(* PLC project CoDeSys External Library Template, WAGO e!COCKPIT e!COCKPIT, author 3S - Smart Software Solutions GmbH *)
(* stored: creationDateTime 2019-10-29T12:22:40.7336323, version 3.5.5.30, modificationDateTime 2019-10-24T14:40:07.960949, organization 3S - Smart Software Solutions GmbH *)
(* Library project template with all possible element types, docu and a sample project structure *)

FUNCTION_BLOCK fbPPPSWezelClimatixPOL63x
  VAR_INPUT
    sKomunikat : alSTRINGKomunikat;  (* komunikat z systemu zewnętrznego *)
    intTablicaKomunikatowRozmiar : INT;  (* rozmiar tablicy danych wysyłkowych *)
    intModbusOdczytZapisZadanieRozmiar : INT;  (* rozmiar tablicy danych modbusa *)
    xTablicaKomunikatowHold : BOOL;  (* wstrzymanie komunikacji mniej ważnych komunikatów *)
    sIdInstancji : STRING;  (* parametr ID rolety np NS02L*202IBM**** *)
    sIdAplikacji : STRING;  (* parametr ID aplikacji np SO*******ECL*000 *)
    sMnemonik : STRING;  (* mnemonik właściciela - BCB* *)
    sMACAdres : STRING;  (* MAC adres sterownika *)
    sDaneZapasowe : STRING;  (* 6 znaków zapasu *)
    tCzasOpoznieniaRestartu : TIME;  (* czas opóźnienia po którym zaczynają być raportowane wartości *)
    tCzasOpoznieniaAlarmu : TIME := TIME#1m0s0ms;  (* czas opóźnienia po którym zaczynają być raportowane wartości *)
    bAdres : BYTE;
    tMinimalnyCzasRaportowania : TIME;
    tMaksymalnyCzasRaportowania : TIME;
    xAutonomizacja : BOOL;
    xAutonomizacjaSztuczna : BOOL;
    xSezonGrzewczyCalyRok : BOOL;
    tCzestotliwoscWysylaniaAlternatywnyAlgorytm : TIME;
    wZaprogramowanyTypInstalacji : WORD;
    rKrzywaGrzewczaTemperaturyZewnetrznejX2HC1Autonomizacja : REAL;  (* Sterowanie w trybie autonomizacji *)
    rKrzywaGrzewczaTemperaturyZasilaniaY2HC1Autonomizacja : REAL;
    rKrzywaGrzewczaTemperaturyZewnetrznejX3HC1Autonomizacja : REAL;
    rKrzywaGrzewczaTemperaturyZasilaniaY3HC1Autonomizacja : REAL;
    rKrzywaGrzewczaTemperaturyZewnetrznejX4HC1Autonomizacja : REAL;
    rKrzywaGrzewczaTemperaturyZasilaniaY4HC1Autonomizacja : REAL;
    rKrzywaGrzewczaTemperaturyZewnetrznejX5HC1Autonomizacja : REAL;
    rKrzywaGrzewczaTemperaturyZasilaniaY5HC1Autonomizacja : REAL;
    rKrzywaGrzewczaTemperaturyZewnetrznejX6HC1Autonomizacja : REAL;
    rKrzywaGrzewczaTemperaturyZasilaniaY6HC1Autonomizacja : REAL;
    intTrybPracyDHWAutonomizacja : INT;
  END_VAR
  VAR_IN_OUT
    arModbusOdczytCykliczny : ARRAY[1..5000] OF typModbusOdczytCykliczny;
    arModbusStatusKomunikacji : ARRAY[1..256] OF INT;
    arModbusOdczytZapisZadanie : ARRAY[1..1000] OF typModbusOdczytZapisZadanie;
    intModbusOdczytZapisZadanieZnacznikZapisu : INT;
    arTablicaKomunikatow : alARRAYTablicaKomunikatow;
    intTablicaKomunikatowZnacznikZapisu : INT;
    aTemperatury : ARRAY[0..96] OF REAL;  (* Tablica pomiarów temperatur bieżącego dnia *)
    rTemperaturaSrednia1Dzien : REAL;  (* Średnia dzienna temperatura *)
    iTemperaturyIndex : INT;  (* Index tablicy *)
    aTemperaturySrednie : ARRAY[0..2] OF REAL;  (* Tablica zawierająca średnie temperatury z trzech ostatnich dni *)
    iTemperaturySrednieIndex : INT;  (* Index tablicy śrenich temperatur *)
    rTemperaturaSrednia3Dni : REAL;  (* Średnia temperatura z trzech dni *)
    xTemperaturaSrednia3DniObliczona : BOOL;  (* Prawda, jeśli obliczona została średnia temperatura z trzech dni *)
  END_VAR
  VAR CONSTANT
    uintTrybPracyHC1AdresModbus : UINT := 400;  (* 1 *)
    uintKrzywaGrzewczaTemperaturyZewnetrznejX2HC1AdresModbus : UINT := 424;  (* 2 *)
    uintKrzywaGrzewczaTemperaturyZewnetrznejX3HC1AdresModbus : UINT := 449;  (* 9 *)
    uintKrzywaGrzewczaTemperaturyZewnetrznejX4HC1AdresModbus : UINT := 450;  (* 10 *)
    uintKrzywaGrzewczaTemperaturyZewnetrznejX5HC1AdresModbus : UINT := 451;  (* 11 *)
    uintKrzywaGrzewczaTemperaturyZewnetrznejX6HC1AdresModbus : UINT := 425;  (* 3 *)
    uintKrzywaGrzewczaTemperaturyZasilaniaY2HC1AdresModbus : UINT := 426;  (* 4 *)
    uintKrzywaGrzewczaTemperaturyZasilaniaY3HC1AdresModbus : UINT := 435;  (* 6 *)
    uintKrzywaGrzewczaTemperaturyZasilaniaY4HC1AdresModbus : UINT := 436;  (* 7 *)
    uintKrzywaGrzewczaTemperaturyZasilaniaY5HC1AdresModbus : UINT := 437;  (* 8 *)
    uintKrzywaGrzewczaTemperaturyZasilaniaY6HC1AdresModbus : UINT := 427;  (* 5 *)
    uintTrybPracyZadanieDHWAdresModbus : UINT := 800;  (* 12 *)
  END_VAR
  VAR
    xPierwszySkan : BOOL := TRUE;
    intPetlaPierwszySkan : INT := 1;
    xInstalacjaHC1 : BOOL;  (* Heat circuit 1 - 1-szy obwód grzewczy *)
    xInstalacjaDHW : BOOL;  (* Domestic hot water - ciepła woda użytkowa *)
    xInstalacjaHP : BOOL;  (* ??? - BRAK ZAPROGRAMOWANIA *)
    xInstalacjaHC2 : BOOL;  (* Heat circuit 2 - 2-gi obwód grzewczy - BRAK ZAPROGRAMOWANIA *)
    fbAutonomizacja : R_TRIG;  (* Wykrywanie przejścia w stan autonomizacji *)
    xPrzywrocDomyslne : BOOL;  (* Przywrócenie nastaw krzywej grzewczej i trybów pracy (przepisanie rAutonomizacjaKrzywaGrzewcza[...] etc. do Climatixa) *)
    intBlokadaWykonywaniaRozkazow : INT;
    intBlokadaWykonywaniaRozkazowZaraportowana : INT;
    xOdczytanaKlasaAlarmuBezpieczenstwa : BOOL := FALSE;  (* definicja zmiennych do odczytu wartości z modbusa klasy alarmów *)
    xOdczytanaKlasaAlarmuKrytyczny : BOOL := FALSE;
    xOdczytanaKlasaAlarmuOstrzezenie : BOOL := FALSE;
    xOdczytanaKlasaAlarmuInformacyjny : BOOL := FALSE;
    wAlarmsWord1 : WORD;  (* alarmy *)
    wAlarmsWord1Zaraportowana : WORD;
    wAlarmsWord2 : WORD;
    wAlarmsWord2Zaraportowana : WORD;
    wAlarmsWord3 : WORD;
    wAlarmsWord3Zaraportowana : WORD;
    wAlarmsWord4 : WORD;
    wAlarmsWord4Zaraportowana : WORD;
    wActiveAlarmsClass0 : WORD;
    wActiveAlarmsClass1 : WORD;
    wActiveAlarmsClass2 : WORD;
    wActiveAlarmsClass3 : WORD;
    wReczneWylaczenieInstalacji : WORD;  (* odczyt *)
    xReczneWylaczenieInstalacji : BOOL;
    wTypInstalacji : WORD;  (* 0=Other,1=1 HC,2=1 HC + DHW,3=1 HC + DHW + HP,4=2 HC,5=2 HC + DHW,6=2 HC + DHW + HP,7=Free (other combination) *)
    wTemperaturaZewnetrzna : WORD;  (* HC1 Temperatura zewnętrzna *)
    rTemperaturaZewnetrzna : REAL;
    fbTemperaturaZewnetrzna : fbFiltrWartoscAnalogowa;
    rTemperaturaZewnetrznaZaraportowana : REAL;
    wTemperaturaGrzaniaNastawionaHC1 : WORD;  (* Temperatura nastawiona zasilania *)
    rTemperaturaGrzaniaNastawionaHC1 : REAL;
    fbTemperaturaGrzaniaNastawionaHC1 : fbFiltrWartoscAnalogowa;
    rTemperaturaGrzaniaNastawionaHC1Zaraportowana : REAL;
    wTemperaturaGrzaniaNastawionaKrzywaGrzewczaHC1 : WORD;  (* Temperatura nastawiona zasilania z krzywej grzewczej *)
    rTemperaturaGrzaniaNastawionaKrzywaGrzewczaHC1 : REAL;
    fbTemperaturaGrzaniaNastawionaKrzywaGrzewczaHC1 : fbFiltrWartoscAnalogowa;
    rTemperaturaGrzaniaNastawionaKrzywaGrzewczaHC1Zaraportowana : REAL;
    wTrybPracyHC1 : WORD;  (* Tryb Pracy *)
    intTrybPracyHC1 : INT;
    intTrybPracyHC1Zaraportowana : INT;
    intTrybPracyHC1Autonomizacja : INT;
    wTrybPracyHC1Ramka : WORD;
    xTrybPracyHC1Zapisz : BOOL;  (* Trigger zapisu wartości w pamięci urządzenia *)
    rTrybPracyHC1Zapis : REAL;  (* Wartość do zapisania w pamięci urządzenia *)
    wTrybOperacjiHC1 : WORD;  (* Tryb operacji *)
    intTrybOperacjiHC1 : INT;
    intTrybOperacjiHC1Zaraportowana : INT;
    wTemperaturaZasilaniaObwoduHC1 : WORD;  (* Obwód na instalację *)
    rTemperaturaZasilaniaObwoduHC1 : REAL;
    fbTemperaturaZasilaniaObwoduHC1 : fbFiltrWartoscAnalogowa;
    rTemperaturaZasilaniaObwoduHC1Zaraportowana : REAL;
    wTemperaturaPowrotuObwoduHC1 : WORD;  (* Obwód na instalację *)
    rTemperaturaPowrotuObwoduHC1 : REAL;
    fbTemperaturaPowrotuObwoduHC1 : fbFiltrWartoscAnalogowa;
    rTemperaturaPowrotuObwoduHC1Zaraportowana : REAL;
    wTemperaturaPowrotuMiastoHC1 : WORD;  (* Powrót przy wymienniku ciepła po stronie wyskoiego parametru (miejskiej sieci ciepłowniczej) *)
    rTemperaturaPowrotuMiastoHC1 : REAL;
    fbTemperaturaPowrotuMiastoHC1 : fbFiltrWartoscAnalogowa;
    rTemperaturaPowrotuMiastoHC1Zaraportowana : REAL;
    wTemperaturaZasilaniaBudynku : WORD;  (* Zasilanie przy wymienniku ciepła po stronie budynku *)
    rTemperaturaZasilaniaBudynku : REAL;
    fbTemperaturaZasilaniaBudynku : fbFiltrWartoscAnalogowa;
    rTemperaturaZasilaniaBudynkuZaraportowana : REAL;
    wTemperaturaPowrotuBudynku : WORD;  (* Powrót przy wymienniku ciepła po stronie budynku *)
    rTemperaturaPowrotuBudynku : REAL;
    fbTemperaturaPowrotuBudynku : fbFiltrWartoscAnalogowa;
    rTemperaturaPowrotuBudynkuZaraportowana : REAL;
    wSygnalZadaniaGrzaniaHC1 : WORD;  (* Sygnał żądanego grzania, w procentach *)
    rSygnalZadaniaGrzaniaHC1 : REAL;
    fbSygnalZadaniaGrzaniaHC1 : fbFiltrWartoscAnalogowa;
    rSygnalZadaniaGrzaniaHC1Zaraportowana : REAL;
    wStopienOtwarciaZaworuMiastoHC1 : WORD;  (* Stopień otwarcia zaworu na powrocie wymiennika po stronie miejskiej sieci ciepłowniczej *)
    rStopienOtwarciaZaworuMiastoHC1 : REAL;
    fbStopienOtwarciaZaworuMiastoHC1 : fbFiltrWartoscAnalogowa;
    rStopienOtwarciaZaworuMiastoHC1Zaraportowana : REAL;
    wKrzywaGrzewczaTemperaturyZewnetrznejX2OdczytHC1 : WORD;  (* Krzywa grzewcza X2 *)
    rKrzywaGrzewczaTemperaturyZewnetrznejX2HC1 : REAL;
    fbKrzywaGrzewczaTemperaturyZewnetrznejX2HC1 : fbFiltrWartoscAnalogowa;
    rKrzywaGrzewczaTemperaturyZewnetrznejX2HC1Zaraportowana : REAL;
    xKrzywaGrzewczaTemperaturyZewnetrznejX2HC1Zapisz : BOOL;  (* Trigger zapisu wartości w pamięci urządzenia *)
    rKrzywaGrzewczaTemperaturyZewnetrznejX2HC1Zapis : REAL;  (* Wartość do zapisania w pamięci urządzenia *)
    wKrzywaGrzewczaTemperaturyZewnetrznejX2HC1Zapis : WORD;  (* Wartość do zapisania w pamięci urządzenia (po konwersji na WORDa) *)
    rKrzywaGrzewczaTemperaturyZewnetrznejX2HC1Raport : REAL;  (* Wartość do zaraportowania *)
    wKrzywaGrzewczaTemperaturyZasilaniaY2OdczytHC1 : WORD;  (* Krzywa grzewcza Y2 *)
    rKrzywaGrzewczaTemperaturyZasilaniaY2HC1 : REAL;
    fbKrzywaGrzewczaTemperaturyZasilaniaY2HC1 : fbFiltrWartoscAnalogowa;
    rKrzywaGrzewczaTemperaturyZasilaniaY2HC1Zaraportowana : REAL;
    xKrzywaGrzewczaTemperaturyZasilaniaY2HC1Zapisz : BOOL;  (* Trigger zapisu wartości w pamięci urządzenia *)
    rKrzywaGrzewczaTemperaturyZasilaniaY2HC1Zapis : REAL;  (* Wartość do zapisania w pamięci urządzenia *)
    wKrzywaGrzewczaTemperaturyZewnetrznejX3OdczytHC1 : WORD;  (* Krzywa grzewcza X3 *)
    rKrzywaGrzewczaTemperaturyZewnetrznejX3HC1 : REAL;
    fbKrzywaGrzewczaTemperaturyZewnetrznejX3HC1 : fbFiltrWartoscAnalogowa;
    rKrzywaGrzewczaTemperaturyZewnetrznejX3HC1Zaraportowana : REAL;
    xKrzywaGrzewczaTemperaturyZewnetrznejX3HC1Zapisz : BOOL;  (* Trigger zapisu wartości w pamięci urządzenia *)
    rKrzywaGrzewczaTemperaturyZewnetrznejX3HC1Zapis : REAL;  (* Wartość do zapisania w pamięci urządzenia *)
    wKrzywaGrzewczaTemperaturyZewnetrznejX3HC1Zapis : WORD;  (* Wartość do zapisania w pamięci urządzenia (po konwersji na WORDa) *)
    rKrzywaGrzewczaTemperaturyZewnetrznejX3HC1Raport : REAL;  (* Wartość do zaraportowania *)
    wKrzywaGrzewczaTemperaturyZasilaniaY3OdczytHC1 : WORD;  (* Krzywa grzewcza Y3 *)
    rKrzywaGrzewczaTemperaturyZasilaniaY3HC1 : REAL;
    fbKrzywaGrzewczaTemperaturyZasilaniaY3HC1 : fbFiltrWartoscAnalogowa;
    rKrzywaGrzewczaTemperaturyZasilaniaY3HC1Zaraportowana : REAL;
    xKrzywaGrzewczaTemperaturyZasilaniaY3HC1Zapisz : BOOL;  (* Trigger zapisu wartości w pamięci urządzenia *)
    rKrzywaGrzewczaTemperaturyZasilaniaY3HC1Zapis : REAL;  (* Wartość do zapisania w pamięci urządzenia *)
    wKrzywaGrzewczaTemperaturyZewnetrznejX4OdczytHC1 : WORD;  (* Krzywa grzewcza X4 *)
    rKrzywaGrzewczaTemperaturyZewnetrznejX4HC1 : REAL;
    fbKrzywaGrzewczaTemperaturyZewnetrznejX4HC1 : fbFiltrWartoscAnalogowa;
    rKrzywaGrzewczaTemperaturyZewnetrznejX4HC1Zaraportowana : REAL;
    xKrzywaGrzewczaTemperaturyZewnetrznejX4HC1Zapisz : BOOL;  (* Trigger zapisu wartości w pamięci urządzenia *)
    rKrzywaGrzewczaTemperaturyZewnetrznejX4HC1Zapis : REAL;  (* Wartość do zapisania w pamięci urządzenia *)
    wKrzywaGrzewczaTemperaturyZewnetrznejX4HC1Zapis : WORD;  (* Wartość do zapisania w pamięci urządzenia (po konwersji na WORDa) *)
    rKrzywaGrzewczaTemperaturyZewnetrznejX4HC1Raport : REAL;  (* Wartość do zaraportowania *)
    wKrzywaGrzewczaTemperaturyZasilaniaY4OdczytHC1 : WORD;  (* Krzywa grzewcza Y4 *)
    rKrzywaGrzewczaTemperaturyZasilaniaY4HC1 : REAL;
    fbKrzywaGrzewczaTemperaturyZasilaniaY4HC1 : fbFiltrWartoscAnalogowa;
    rKrzywaGrzewczaTemperaturyZasilaniaY4HC1Zaraportowana : REAL;
    xKrzywaGrzewczaTemperaturyZasilaniaY4HC1Zapisz : BOOL;  (* Trigger zapisu wartości w pamięci urządzenia *)
    rKrzywaGrzewczaTemperaturyZasilaniaY4HC1Zapis : REAL;  (* Wartość do zapisania w pamięci urządzenia *)
    wKrzywaGrzewczaTemperaturyZewnetrznejX5OdczytHC1 : WORD;  (* Krzywa grzewcza X5 *)
    rKrzywaGrzewczaTemperaturyZewnetrznejX5HC1 : REAL;
    fbKrzywaGrzewczaTemperaturyZewnetrznejX5HC1 : fbFiltrWartoscAnalogowa;
    rKrzywaGrzewczaTemperaturyZewnetrznejX5HC1Zaraportowana : REAL;
    xKrzywaGrzewczaTemperaturyZewnetrznejX5HC1Zapisz : BOOL;  (* Trigger zapisu wartości w pamięci urządzenia *)
    rKrzywaGrzewczaTemperaturyZewnetrznejX5HC1Zapis : REAL;  (* Wartość do zapisania w pamięci urządzenia *)
    wKrzywaGrzewczaTemperaturyZewnetrznejX5HC1Zapis : WORD;  (* Wartość do zapisania w pamięci urządzenia (po konwersji na WORDa) *)
    rKrzywaGrzewczaTemperaturyZewnetrznejX5HC1Raport : REAL;  (* Wartość do zaraportowania *)
    wKrzywaGrzewczaTemperaturyZasilaniaY5OdczytHC1 : WORD;  (* Krzywa grzewcza Y5 *)
    rKrzywaGrzewczaTemperaturyZasilaniaY5HC1 : REAL;
    fbKrzywaGrzewczaTemperaturyZasilaniaY5HC1 : fbFiltrWartoscAnalogowa;
    rKrzywaGrzewczaTemperaturyZasilaniaY5HC1Zaraportowana : REAL;
    xKrzywaGrzewczaTemperaturyZasilaniaY5HC1Zapisz : BOOL;  (* Trigger zapisu wartości w pamięci urządzenia *)
    rKrzywaGrzewczaTemperaturyZasilaniaY5HC1Zapis : REAL;  (* Wartość do zapisania w pamięci urządzenia *)
    wKrzywaGrzewczaTemperaturyZewnetrznejX6OdczytHC1 : WORD;  (* Krzywa grzewcza X6 *)
    rKrzywaGrzewczaTemperaturyZewnetrznejX6HC1 : REAL;
    fbKrzywaGrzewczaTemperaturyZewnetrznejX6HC1 : fbFiltrWartoscAnalogowa;
    rKrzywaGrzewczaTemperaturyZewnetrznejX6HC1Zaraportowana : REAL;
    xKrzywaGrzewczaTemperaturyZewnetrznejX6HC1Zapisz : BOOL;  (* Trigger zapisu wartości w pamięci urządzenia *)
    rKrzywaGrzewczaTemperaturyZewnetrznejX6HC1Zapis : REAL;  (* Wartość do zapisania w pamięci urządzenia *)
    wKrzywaGrzewczaTemperaturyZewnetrznejX6HC1Zapis : WORD;  (* Wartość do zapisania w pamięci urządzenia (po konwersji na WORDa) *)
    rKrzywaGrzewczaTemperaturyZewnetrznejX6HC1Raport : REAL;  (* Wartość do zaraportowania *)
    wKrzywaGrzewczaTemperaturyZasilaniaY6OdczytHC1 : WORD;  (* Krzywa grzewcza Y6 *)
    rKrzywaGrzewczaTemperaturyZasilaniaY6HC1 : REAL;
    fbKrzywaGrzewczaTemperaturyZasilaniaY6HC1 : fbFiltrWartoscAnalogowa;
    rKrzywaGrzewczaTemperaturyZasilaniaY6HC1Zaraportowana : REAL;
    xKrzywaGrzewczaTemperaturyZasilaniaY6HC1Zapisz : BOOL;  (* Trigger zapisu wartości w pamięci urządzenia *)
    rKrzywaGrzewczaTemperaturyZasilaniaY6HC1Zapis : REAL;  (* Wartość do zapisania w pamięci urządzenia *)
    wTemperaturaGrzaniaNastawionaDHW : WORD;  (* DHW Temperatura nastawiona zasilania *)
    rTemperaturaGrzaniaNastawionaDHW : REAL;
    fbTemperaturaGrzaniaNastawionaDHW : fbFiltrWartoscAnalogowa;
    rTemperaturaGrzaniaNastawionaDHWZaraportowana : REAL;
    wTrybPracyDHW : WORD;  (* Tryb Pracy *)
    intTrybPracyDHW : INT;
    intTrybPracyDHWZaraportowana : INT;
    wTrybPracyDHWRamka : WORD;
    xTrybPracyDHWZapisz : BOOL;  (* Trigger zapisu wartości w pamięci urządzenia *)
    rTrybPracyDHWZapis : REAL;  (* Wartość do zapisania w pamięci urządzenia *)
    wTrybOperacjiDHW : WORD;  (* Tryb operacji *)
    intTrybOperacjiDHW : INT;
    intTrybOperacjiDHWZaraportowana : INT;
    wTemperaturaPowrotuMiastoDHW : WORD;  (* Powrót przy wymienniku ciepła po stronie wyskoiego parametru (miejskiej sieci ciepłowniczej) *)
    rTemperaturaPowrotuMiastoDHW : REAL;
    fbTemperaturaPowrotuMiastoDHW : fbFiltrWartoscAnalogowa;
    rTemperaturaPowrotuMiastoDHWZaraportowana : REAL;
    wTemperaturaZasilaniaBudynekDHW : WORD;  (* Zasilanie przy wymienniku ciepła po stronie budynku *)
    rTemperaturaZasilaniaBudynekDHW : REAL;
    fbTemperaturaZasilaniaBudynekDHW : fbFiltrWartoscAnalogowa;
    rTemperaturaZasilaniaBudynekDHWZaraportowana : REAL;
    wTemperaturaPowrotuBudynekDHW : WORD;  (* Powrót przy wymienniku ciepła po stronie budynku *)
    rTemperaturaPowrotuBudynekDHW : REAL;
    fbTemperaturaPowrotuBudynekDHW : fbFiltrWartoscAnalogowa;
    rTemperaturaPowrotuBudynekDHWZaraportowana : REAL;
    wStopienOtwarciaZaworuMiastoDHW : WORD;  (* Stopień otwarcia zaworu na powrocie wymiennika po stronie miejskiej sieci ciepłowniczej *)
    rStopienOtwarciaZaworuMiastoDHW : REAL;
    fbStopienOtwarciaZaworuMiastoDHW : fbFiltrWartoscAnalogowa;
    rStopienOtwarciaZaworuMiastoDHWZaraportowana : REAL;
    xPoInicjalizacji : BOOL := FALSE;  (* inicjalizacja *)
    fbInicjalizacyjnyTimer : TON;
    tCzasInicjalizacji : TIME := TIME#30s0ms;
    sDane : alSTRINGKomunikat;  (* pozostale definicje *)
    sWyslanyKomunikatDummy : alSTRINGKomunikat;
    xZadanieRaportu : BOOL;
    sKomunikatPamiec : alSTRINGKomunikat;
    intPetla : INT;
    arErrorStan : ARRAY[0..11] OF INT;  (* tablica przechowująca statusy alarmowe *)
    arErrorKlasa : ARRAY[0..11] OF INT;  (* tablica przechowująca klasy danych alarmów *)
    xRaport : BOOL := FALSE;
    sTempWartoscAtrybutu : STRING;
    xOverFlow : BOOL;
    rtrigPrzywrocDomyslne : R_TRIG;  (* Przywracanie domyślnych wartości nastaw *)
    rtrigZapisModbus : R_TRIG;  (* Triger zapisu danych po Modbusie *)
    fbTaktowanieZapisywaniaModbus : TON;  (* Cykliczne żądanie zapisu danych do urządzenia *)
    fbTimerBrakuKomunikacji : TON;  (* Kontrola komunikacji urządzenia *)
    xBrakKomunikacjiPLC : BOOL;
    xBrakKomunikacjiIZE : BOOL;
    wTrybPracyZadanie : INT;
    rAutonomizacjaKorektaTemperaturyGrzaniaZadanie : INT;
    xBrakKomunikacji : BOOL;
    rTemperaturaZewnetrznaPamiec : REAL;  (* Sprawdzanie sprawności czujnika temperatury zewnętrznej *)
    xBrakZmianyTemperaturyZewnetrznej : BOOL;
    fbBrakZmianyTemperaturyZewnetrznejTimer : TON;
    xBladBrakZmianyTemperaturyZewnetrznej : BOOL;
    rTemperaturaZasilaniaObwoduHC1Pamiec : REAL;  (* Sprawdzanie sprawności czujnika temperatury zasilania obwodu HC1 *)
    xBrakZmianyTemperaturyZasilaniaObwoduHC1 : BOOL;
    fbBrakZmianyTemperaturyZasilaniaObwoduHC1Timer : TON;
    xBladBrakZmianyTemperaturyZasilaniaObwoduHC1 : BOOL;
    rTemperaturaZasilaniaObwoduDHWPamiec : REAL;  (* Sprawdzanie sprawności czujnika temperatury zasilania obwodu DHW *)
    xBrakZmianyTemperaturyZasilaniaObwoduDHW : BOOL;
    fbBrakZmianyTemperaturyZasilaniaObwoduDHWTimer : TON;
    xBladBrakZmianyTemperaturyZasilaniaObwoduDHW : BOOL;
    xBrakOsiagnieciaTemperauryZadanejHC1 : BOOL;  (* Sprawdzanie czy została osiągnęta zadana temperatura zasilania obwodu HC1 *)
    fbBrakOsiagnieciaTemperauryZadanejHC1Timer : TON;
    xBladBrakOsiagnieciaTemperauryZadanejHC1 : BOOL;
    xBrakOsiagnieciaTemperauryZadanejDHW : BOOL;  (* Sprawdzanie czy została osiągnęta zadana temperatura zasilania obwodu DHW *)
    fbBrakOsiagnieciaTemperauryZadanejDHWTimer : TON;
    xBladBrakOsiagnieciaTemperauryZadanejDHW : BOOL;
    fbWschodZachod : FbCalculateSunriseSunset;  (* Obliczanie wschodu i zachodu słońca *)
    fbZegar15M : TON;  (* Timer taktujący zapisywanie temperatury *)
    xObliczSrednia3Dni : BOOL;  (* Triger obliczania średniej dziennej temperatury z 3 ostatnich dni *)
    iIloscPomiarow : INT;  (* Ilość pomiarów dokonanych w ciągu dnia *)
    rTemperaturaSrednia1DzienZaraportowana : REAL;  (* Średnia dzienna temperatura zaraporotawana *)
    xSezonGrzewczy : BOOL;  (* Włączenie ogrzewania *)
    xSezonGrzewczyZaraportowana : BOOL;  (* Włączenie ogrzewania zaraportowane *)
    xBladIloscPomiarowTemperatury : BOOL;  (* Zbyt mała ilość pomiarów dokonanych w ciągu dnia do obliczenia średniej *)
  END_VAR

            (*			
Autor:					Paweł Kąkol, 2018-09-03 
Prawa majątkowe: 		Solwena Sp. z o.o., 
Aktualizacje:			2018-09-06-PK: zmiana adresów rejestrów o -1
						2018-09-07-PK: przerobienie całego fb tak aby realizował układ HC1 (1-szego obiegu grzewczego) oraz/lub DHW (ciepłej wody użytkowej), wykonanie reakcji na autonomizację
						2019-01-04-AW: zmiana odczytu klasy alarmów (zmiana funkcji i adresów); odczyt rejestrów zawierających info o rodzaju alarmu
						2019-02-08-AWy: OverFlow
						2019-02-10-AWy: odczyt trybu operacji HC1 i wysyłanie do IZE, poprawa odczytywania i wysyłania temperatury zasilania, powrotu obwodu i miasta, krzywej grzewczej etc.
						2019-02-18-AWy: odczyt trybu operacji DHW i wysyłanie do IZE
						2019-05-15-AWy: - modyfikacja warunku obsługi ramki C. Było: IF sTempWartoscAtrybutu <> '' AND intBlokadaWykonywaniaRozkazow = 0 THEN. Jest: IF intBlokadaWykonywaniaRozkazow = 0 THEN
						2019-05-16-AWy: - modyfikacja warunku ręcznej inizjalizacji trybów pracy i krzywej grzewczej. Było: IF xAutonomizacja THEN. Jest: IF xPrzywrocDomyslne THEN.
									    - modyfikacja warunku na raportowanie. Dopisane: AND xPoInicjalizacji
									    - modyfikacja warunków na zapis po otrzymaniu ramki C. Nowy warunek: IF fnKomunikatDaneSzukajWartosci(sKomunikat,'TEMPKGHC1X5=') <> '' THEN etc.
						2019-05-23-AWy: dodanie przesyłania wewnętrznych numerów błędów z Climatixa (wAlarmsWord1 etc.)
						2019-06-03-AWy: załadowanie domyślnych trybów pracy i nastaw po przejściu w tryb autonomizacji
						2019-06-04-AWy: usunięcie błędów generowanych przy odczycie liczb ujemnych
						2019-07-16-AWy: zmiana typu zmiennej intTrybPracyDHWAutonomizacja z WORD na INT
						2019-08-05-AWy: wyznaczanie okresu grzewczego. Wysyłanie xSezonGrzewczy i rTemperaturaSrednia1Dzien do IZE. Przeniesie xTrybPracyAutonomizacja z VAR_INPUT do VAR
						2019-10-22-AWy: - wydłużenie czasu fbTaktowanieZapisywaniaModbus oraz wprowadzenie trigera zapisu po Modbusie
										- zmiana trigera fbTimerBrakuKomunikacji
						
Opis:					fb służy do komunikacji po Modbus RTU z węzłem ciepła na budynkach ENGIE, gdzie zainstalowano Siemens Climatix POL638.70
						Zawiera kod wykonywany w razie autonomizacji - wysyłanie zmiennych wprowadzonych poprzez EIG,
						po ustaniu Autonomizacji zostaje utrzymany stan z Autonomizacji, a układ reaguje dopiero na nowe ramki

UWAGA:					Zaprogramowano HC1 oraz DHN, nie zaprogramowane HP i HC2 
*)


//inicjalizacja sterownika
fbInicjalizacyjnyTimer(IN := (NOT xPoInicjalizacji AND arModbusStatusKomunikacji[bAdres] = enumModbusStatus.KomunikacjaPrawidlowa) , PT := tCzasOpoznieniaRestartu);
IF fbInicjalizacyjnyTimer.Q THEN
	IF xInstalacjaHC1 OR xInstalacjaHC2 THEN
		rTemperaturaZewnetrznaZaraportowana := rTemperaturaZewnetrzna;
	END_IF
	IF xInstalacjaHC1 THEN
		rTemperaturaGrzaniaNastawionaHC1Zaraportowana := rTemperaturaGrzaniaNastawionaHC1;
		rTemperaturaGrzaniaNastawionaKrzywaGrzewczaHC1Zaraportowana := rTemperaturaGrzaniaNastawionaKrzywaGrzewczaHC1;
		intTrybPracyHC1Zaraportowana := intTrybPracyHC1;
		intTrybOperacjiHC1 := intTrybOperacjiHC1Zaraportowana;
		rTemperaturaZasilaniaObwoduHC1Zaraportowana := rTemperaturaZasilaniaObwoduHC1;
		rTemperaturaPowrotuObwoduHC1Zaraportowana := rTemperaturaPowrotuObwoduHC1;
		rTemperaturaPowrotuMiastoHC1Zaraportowana := rTemperaturaPowrotuMiastoHC1;
		rTemperaturaZasilaniaBudynkuZaraportowana := rTemperaturaZasilaniaBudynku;
		rTemperaturaPowrotuBudynkuZaraportowana := rTemperaturaPowrotuBudynku;
		rSygnalZadaniaGrzaniaHC1Zaraportowana := rSygnalZadaniaGrzaniaHC1;
		rStopienOtwarciaZaworuMiastoHC1Zaraportowana := rStopienOtwarciaZaworuMiastoHC1;
		rKrzywaGrzewczaTemperaturyZewnetrznejX2HC1Zaraportowana := rKrzywaGrzewczaTemperaturyZewnetrznejX2HC1;
		rKrzywaGrzewczaTemperaturyZasilaniaY2HC1Zaraportowana := rKrzywaGrzewczaTemperaturyZasilaniaY2HC1;
		rKrzywaGrzewczaTemperaturyZewnetrznejX3HC1Zaraportowana := rKrzywaGrzewczaTemperaturyZewnetrznejX3HC1;
		rKrzywaGrzewczaTemperaturyZasilaniaY3HC1Zaraportowana := rKrzywaGrzewczaTemperaturyZasilaniaY3HC1;
		rKrzywaGrzewczaTemperaturyZewnetrznejX4HC1Zaraportowana := rKrzywaGrzewczaTemperaturyZewnetrznejX4HC1;
		rKrzywaGrzewczaTemperaturyZasilaniaY4HC1Zaraportowana := rKrzywaGrzewczaTemperaturyZasilaniaY4HC1;
		rKrzywaGrzewczaTemperaturyZewnetrznejX5HC1Zaraportowana := rKrzywaGrzewczaTemperaturyZewnetrznejX5HC1;
		rKrzywaGrzewczaTemperaturyZasilaniaY5HC1Zaraportowana := rKrzywaGrzewczaTemperaturyZasilaniaY5HC1;
		rKrzywaGrzewczaTemperaturyZewnetrznejX6HC1Zaraportowana := rKrzywaGrzewczaTemperaturyZewnetrznejX6HC1;
		rKrzywaGrzewczaTemperaturyZasilaniaY6HC1Zaraportowana := rKrzywaGrzewczaTemperaturyZasilaniaY6HC1;
		xSezonGrzewczyZaraportowana := xSezonGrzewczy;
		rTemperaturaSrednia1DzienZaraportowana := rTemperaturaSrednia1Dzien;
	END_IF
	IF xInstalacjaDHW THEN
		rTemperaturaGrzaniaNastawionaDHWZaraportowana := rTemperaturaGrzaniaNastawionaDHW;
		intTrybPracyDHWZaraportowana := intTrybPracyDHW;
		rTemperaturaPowrotuMiastoDHWZaraportowana := rTemperaturaPowrotuMiastoDHW;
		rTemperaturaZasilaniaBudynekDHWZaraportowana := rTemperaturaZasilaniaBudynekDHW;
		rTemperaturaPowrotuBudynekDHWZaraportowana := rTemperaturaPowrotuBudynekDHW;
		rStopienOtwarciaZaworuMiastoDHWZaraportowana := rStopienOtwarciaZaworuMiastoDHW;
		intTrybOperacjiDHWZaraportowana := intTrybOperacjiDHW;
	END_IF
	wAlarmsWord1Zaraportowana := wAlarmsWord1;
	wAlarmsWord2Zaraportowana := wAlarmsWord2;
	wAlarmsWord3Zaraportowana := wAlarmsWord3;
	wAlarmsWord4Zaraportowana := wAlarmsWord4;
	xPoInicjalizacji := TRUE;
END_IF

// Włącz autonomizację jeśli sterownik jest w stanie inicjalizacji lub nastąpiło wymuszenie autonomizacji
IF NOT xPoInicjalizacji OR xAutonomizacjaSztuczna = TRUE THEN
	xAutonomizacja := TRUE;
END_IF 

// Kontrola komunikacji
fbTimerBrakuKomunikacji(IN := arModbusStatusKomunikacji[bAdres] <> enumModbusStatus.KomunikacjaPrawidlowa, PT := T#60S);
IF fbTimerBrakuKomunikacji.Q THEN
	xBrakKomunikacjiPLC := TRUE;
ELSE
	xBrakKomunikacjiPLC := FALSE;
END_IF

IF xAutonomizacja THEN
	xBrakKomunikacjiIZE := TRUE;
ELSE
	xBrakKomunikacjiIZE := FALSE;
END_IF

// Deklaracja rejestrów Modbusa
IF xPierwszySkan THEN
	xPierwszySkan := FALSE;
	WHILE arModbusOdczytCykliczny[intPetlaPierwszySkan].bAdresUrzadzenia <> 0 DO
		intPetlaPierwszySkan := intPetlaPierwszySkan + 1;
	END_WHILE
	
	//wybrana instalacja na budynku
	CASE wZaprogramowanyTypInstalacji OF
		0:	xInstalacjaHC1 := FALSE;
			xInstalacjaDHW := FALSE;
			xInstalacjaHP := FALSE;
			xInstalacjaHC2 := FALSE;
		1:	xInstalacjaHC1 := TRUE;
			xInstalacjaDHW := FALSE;
			xInstalacjaHP := FALSE;
			xInstalacjaHC2 := FALSE;
		2:	xInstalacjaHC1 := TRUE;
			xInstalacjaDHW := TRUE;
			xInstalacjaHP := FALSE;
			xInstalacjaHC2 := FALSE;
		3:	xInstalacjaHC1 := TRUE;
			xInstalacjaDHW := TRUE;
			xInstalacjaHP := TRUE;
			xInstalacjaHC2 := FALSE;
		4:	xInstalacjaHC1 := TRUE;
			xInstalacjaDHW := FALSE;
			xInstalacjaHP := FALSE;
			xInstalacjaHC2 := TRUE;
		5:	xInstalacjaHC1 := TRUE;
			xInstalacjaDHW := TRUE;
			xInstalacjaHP := FALSE;
			xInstalacjaHC2 := TRUE;
		6:	xInstalacjaHC1 := TRUE;
			xInstalacjaDHW := TRUE;
			xInstalacjaHP := TRUE;
			xInstalacjaHC2 := TRUE;
	END_CASE
	
//deklaracja rejestrow do odczytu
	// Rejestry zawierające informację alarmach
	arModbusOdczytCykliczny[intPetlaPierwszySkan].bAdresUrzadzenia := bAdres;
	arModbusOdczytCykliczny[intPetlaPierwszySkan].bFunkcja := TO_BYTE(enumModbusKodyFunkcji.OdczytNRejestrowWejsciowych);
	arModbusOdczytCykliczny[intPetlaPierwszySkan].uiAdresRejestru := 18;
	arModbusOdczytCykliczny[intPetlaPierwszySkan].ltCzestotliwosc := LTIME#10S;
	arModbusOdczytCykliczny[intPetlaPierwszySkan].pZmiennaReferencyjna := ADR(wAlarmsWord1);
	intPetlaPierwszySkan := intPetlaPierwszySkan + 1;
	
	arModbusOdczytCykliczny[intPetlaPierwszySkan].bAdresUrzadzenia := bAdres;
	arModbusOdczytCykliczny[intPetlaPierwszySkan].bFunkcja := TO_BYTE(enumModbusKodyFunkcji.OdczytNRejestrowWejsciowych);
	arModbusOdczytCykliczny[intPetlaPierwszySkan].uiAdresRejestru := 19;
	arModbusOdczytCykliczny[intPetlaPierwszySkan].ltCzestotliwosc := LTIME#10S;
	arModbusOdczytCykliczny[intPetlaPierwszySkan].pZmiennaReferencyjna := ADR(wAlarmsWord2);
	intPetlaPierwszySkan := intPetlaPierwszySkan + 1;
	
	arModbusOdczytCykliczny[intPetlaPierwszySkan].bAdresUrzadzenia := bAdres;
	arModbusOdczytCykliczny[intPetlaPierwszySkan].bFunkcja := TO_BYTE(enumModbusKodyFunkcji.OdczytNRejestrowWejsciowych);
	arModbusOdczytCykliczny[intPetlaPierwszySkan].uiAdresRejestru := 20;
	arModbusOdczytCykliczny[intPetlaPierwszySkan].ltCzestotliwosc := LTIME#10S;
	arModbusOdczytCykliczny[intPetlaPierwszySkan].pZmiennaReferencyjna := ADR(wAlarmsWord3);
	intPetlaPierwszySkan := intPetlaPierwszySkan + 1;
	
	arModbusOdczytCykliczny[intPetlaPierwszySkan].bAdresUrzadzenia := bAdres;
	arModbusOdczytCykliczny[intPetlaPierwszySkan].bFunkcja := TO_BYTE(enumModbusKodyFunkcji.OdczytNRejestrowWejsciowych);
	arModbusOdczytCykliczny[intPetlaPierwszySkan].uiAdresRejestru := 21;
	arModbusOdczytCykliczny[intPetlaPierwszySkan].ltCzestotliwosc := LTIME#10S;
	arModbusOdczytCykliczny[intPetlaPierwszySkan].pZmiennaReferencyjna := ADR(wAlarmsWord4);
	intPetlaPierwszySkan := intPetlaPierwszySkan + 1;
	
	arModbusOdczytCykliczny[intPetlaPierwszySkan].bAdresUrzadzenia := bAdres;
	arModbusOdczytCykliczny[intPetlaPierwszySkan].bFunkcja := TO_BYTE(enumModbusKodyFunkcji.OdczytNRejestrowWejsciowych);
	arModbusOdczytCykliczny[intPetlaPierwszySkan].uiAdresRejestru := 22;
	arModbusOdczytCykliczny[intPetlaPierwszySkan].ltCzestotliwosc := LTIME#10S;
	arModbusOdczytCykliczny[intPetlaPierwszySkan].pZmiennaReferencyjna := ADR(wActiveAlarmsClass0);
	intPetlaPierwszySkan := intPetlaPierwszySkan + 1;
	
	arModbusOdczytCykliczny[intPetlaPierwszySkan].bAdresUrzadzenia := bAdres;
	arModbusOdczytCykliczny[intPetlaPierwszySkan].bFunkcja := TO_BYTE(enumModbusKodyFunkcji.OdczytNRejestrowWejsciowych);
	arModbusOdczytCykliczny[intPetlaPierwszySkan].uiAdresRejestru := 23;
	arModbusOdczytCykliczny[intPetlaPierwszySkan].ltCzestotliwosc := LTIME#10S;
	arModbusOdczytCykliczny[intPetlaPierwszySkan].pZmiennaReferencyjna := ADR(wActiveAlarmsClass1);
	intPetlaPierwszySkan := intPetlaPierwszySkan + 1;
	
	arModbusOdczytCykliczny[intPetlaPierwszySkan].bAdresUrzadzenia := bAdres;
	arModbusOdczytCykliczny[intPetlaPierwszySkan].bFunkcja := TO_BYTE(enumModbusKodyFunkcji.OdczytNRejestrowWejsciowych);
	arModbusOdczytCykliczny[intPetlaPierwszySkan].uiAdresRejestru := 24;
	arModbusOdczytCykliczny[intPetlaPierwszySkan].ltCzestotliwosc := LTIME#10S;
	arModbusOdczytCykliczny[intPetlaPierwszySkan].pZmiennaReferencyjna := ADR(wActiveAlarmsClass2);
	intPetlaPierwszySkan := intPetlaPierwszySkan + 1;
	
	arModbusOdczytCykliczny[intPetlaPierwszySkan].bAdresUrzadzenia := bAdres;
	arModbusOdczytCykliczny[intPetlaPierwszySkan].bFunkcja := TO_BYTE(enumModbusKodyFunkcji.OdczytNRejestrowWejsciowych);
	arModbusOdczytCykliczny[intPetlaPierwszySkan].uiAdresRejestru := 25;
	arModbusOdczytCykliczny[intPetlaPierwszySkan].ltCzestotliwosc := LTIME#10S;
	arModbusOdczytCykliczny[intPetlaPierwszySkan].pZmiennaReferencyjna := ADR(wActiveAlarmsClass3);
	intPetlaPierwszySkan := intPetlaPierwszySkan + 1;
	
	// Flagi typów alarmów (nie ma pewności, że działa - najprawdopodobniej w dokumentacji jest błąd i typy alarmów to nie inputy a coile - do zweryfikowania) - CAŁOŚĆ DO PRZETESTOWANIA
	arModbusOdczytCykliczny[intPetlaPierwszySkan].bAdresUrzadzenia := bAdres;
	arModbusOdczytCykliczny[intPetlaPierwszySkan].bFunkcja := TO_BYTE(enumModbusKodyFunkcji.OdczytWyjscBitowych);
	arModbusOdczytCykliczny[intPetlaPierwszySkan].uiAdresRejestru := 0;
	arModbusOdczytCykliczny[intPetlaPierwszySkan].ltCzestotliwosc := LTIME#10S;
	arModbusOdczytCykliczny[intPetlaPierwszySkan].pZmiennaReferencyjna := ADR(xOdczytanaKlasaAlarmuBezpieczenstwa);
	intPetlaPierwszySkan := intPetlaPierwszySkan + 1;		
	
	arModbusOdczytCykliczny[intPetlaPierwszySkan].bAdresUrzadzenia := bAdres;
	arModbusOdczytCykliczny[intPetlaPierwszySkan].bFunkcja := TO_BYTE(enumModbusKodyFunkcji.OdczytWyjscBitowych);
	arModbusOdczytCykliczny[intPetlaPierwszySkan].uiAdresRejestru := 1;
	arModbusOdczytCykliczny[intPetlaPierwszySkan].ltCzestotliwosc := LTIME#10S;
	arModbusOdczytCykliczny[intPetlaPierwszySkan].pZmiennaReferencyjna := ADR(xOdczytanaKlasaAlarmuKrytyczny);
	intPetlaPierwszySkan := intPetlaPierwszySkan + 1;	
	
	arModbusOdczytCykliczny[intPetlaPierwszySkan].bAdresUrzadzenia := bAdres;
	arModbusOdczytCykliczny[intPetlaPierwszySkan].bFunkcja := TO_BYTE(enumModbusKodyFunkcji.OdczytWyjscBitowych);
	arModbusOdczytCykliczny[intPetlaPierwszySkan].uiAdresRejestru := 2;
	arModbusOdczytCykliczny[intPetlaPierwszySkan].ltCzestotliwosc := LTIME#10S;
	arModbusOdczytCykliczny[intPetlaPierwszySkan].pZmiennaReferencyjna := ADR(xOdczytanaKlasaAlarmuOstrzezenie);
	intPetlaPierwszySkan := intPetlaPierwszySkan + 1;	
	
	arModbusOdczytCykliczny[intPetlaPierwszySkan].bAdresUrzadzenia := bAdres;
	arModbusOdczytCykliczny[intPetlaPierwszySkan].bFunkcja := TO_BYTE(enumModbusKodyFunkcji.OdczytWyjscBitowych);
	arModbusOdczytCykliczny[intPetlaPierwszySkan].uiAdresRejestru := 3;
	arModbusOdczytCykliczny[intPetlaPierwszySkan].ltCzestotliwosc := LTIME#10S;
	arModbusOdczytCykliczny[intPetlaPierwszySkan].pZmiennaReferencyjna := ADR(xOdczytanaKlasaAlarmuInformacyjny);
	intPetlaPierwszySkan := intPetlaPierwszySkan + 1;
	
	//input register
	arModbusOdczytCykliczny[intPetlaPierwszySkan].bAdresUrzadzenia := bAdres;
	arModbusOdczytCykliczny[intPetlaPierwszySkan].bFunkcja := TO_BYTE(enumModbusKodyFunkcji.OdczytNRejestrowWejsciowych);
	arModbusOdczytCykliczny[intPetlaPierwszySkan].uiAdresRejestru := 4;
	arModbusOdczytCykliczny[intPetlaPierwszySkan].ltCzestotliwosc := TIME_TO_LTIME(tMinimalnyCzasRaportowania);
	arModbusOdczytCykliczny[intPetlaPierwszySkan].pZmiennaReferencyjna := ADR(wReczneWylaczenieInstalacji);
	intPetlaPierwszySkan := intPetlaPierwszySkan + 1;

	arModbusOdczytCykliczny[intPetlaPierwszySkan].bAdresUrzadzenia := bAdres;
	arModbusOdczytCykliczny[intPetlaPierwszySkan].bFunkcja := TO_BYTE(enumModbusKodyFunkcji.OdczytNRejestrowWejsciowych);
	arModbusOdczytCykliczny[intPetlaPierwszySkan].uiAdresRejestru := 9;
	arModbusOdczytCykliczny[intPetlaPierwszySkan].ltCzestotliwosc := TIME_TO_LTIME(tMinimalnyCzasRaportowania);
	arModbusOdczytCykliczny[intPetlaPierwszySkan].pZmiennaReferencyjna := ADR(wTypInstalacji);
	intPetlaPierwszySkan := intPetlaPierwszySkan + 1;
	
	arModbusOdczytCykliczny[intPetlaPierwszySkan].bAdresUrzadzenia := bAdres;
	arModbusOdczytCykliczny[intPetlaPierwszySkan].bFunkcja := TO_BYTE(enumModbusKodyFunkcji.OdczytNRejestrowWejsciowych);
	arModbusOdczytCykliczny[intPetlaPierwszySkan].uiAdresRejestru := 49;
	arModbusOdczytCykliczny[intPetlaPierwszySkan].ltCzestotliwosc := TIME_TO_LTIME(tMinimalnyCzasRaportowania);
	arModbusOdczytCykliczny[intPetlaPierwszySkan].pZmiennaReferencyjna := ADR(wTemperaturaZewnetrzna);
	intPetlaPierwszySkan := intPetlaPierwszySkan + 1;
	
	arModbusOdczytCykliczny[intPetlaPierwszySkan].bAdresUrzadzenia := bAdres;
	arModbusOdczytCykliczny[intPetlaPierwszySkan].bFunkcja := TO_BYTE(enumModbusKodyFunkcji.OdczytNRejestrowWejsciowych);
	arModbusOdczytCykliczny[intPetlaPierwszySkan].uiAdresRejestru := 50;
	arModbusOdczytCykliczny[intPetlaPierwszySkan].ltCzestotliwosc := TIME_TO_LTIME(tMinimalnyCzasRaportowania);
	arModbusOdczytCykliczny[intPetlaPierwszySkan].pZmiennaReferencyjna := ADR(wTemperaturaZasilaniaBudynku);
	intPetlaPierwszySkan := intPetlaPierwszySkan + 1;
	
	arModbusOdczytCykliczny[intPetlaPierwszySkan].bAdresUrzadzenia := bAdres;
	arModbusOdczytCykliczny[intPetlaPierwszySkan].bFunkcja := TO_BYTE(enumModbusKodyFunkcji.OdczytNRejestrowWejsciowych);
	arModbusOdczytCykliczny[intPetlaPierwszySkan].uiAdresRejestru := 51;
	arModbusOdczytCykliczny[intPetlaPierwszySkan].ltCzestotliwosc := TIME_TO_LTIME(tMinimalnyCzasRaportowania);
	arModbusOdczytCykliczny[intPetlaPierwszySkan].pZmiennaReferencyjna := ADR(wTemperaturaPowrotuBudynku);
	intPetlaPierwszySkan := intPetlaPierwszySkan + 1;
	
	IF xInstalacjaHC1 THEN
		arModbusOdczytCykliczny[intPetlaPierwszySkan].bAdresUrzadzenia := bAdres;
		arModbusOdczytCykliczny[intPetlaPierwszySkan].bFunkcja := TO_BYTE(enumModbusKodyFunkcji.OdczytNRejestrowWejsciowych);
		arModbusOdczytCykliczny[intPetlaPierwszySkan].uiAdresRejestru := 449;
		arModbusOdczytCykliczny[intPetlaPierwszySkan].ltCzestotliwosc := TIME_TO_LTIME(tMinimalnyCzasRaportowania);
		arModbusOdczytCykliczny[intPetlaPierwszySkan].pZmiennaReferencyjna := ADR(wTemperaturaZasilaniaObwoduHC1);
		intPetlaPierwszySkan := intPetlaPierwszySkan + 1;
	END_IF
	
	IF xInstalacjaHC1 THEN
		arModbusOdczytCykliczny[intPetlaPierwszySkan].bAdresUrzadzenia := bAdres;
		arModbusOdczytCykliczny[intPetlaPierwszySkan].bFunkcja := TO_BYTE(enumModbusKodyFunkcji.OdczytNRejestrowWejsciowych);
		arModbusOdczytCykliczny[intPetlaPierwszySkan].uiAdresRejestru := 450;
		arModbusOdczytCykliczny[intPetlaPierwszySkan].ltCzestotliwosc := TIME_TO_LTIME(tMinimalnyCzasRaportowania);
		arModbusOdczytCykliczny[intPetlaPierwszySkan].pZmiennaReferencyjna := ADR(wTemperaturaPowrotuObwoduHC1);
		intPetlaPierwszySkan := intPetlaPierwszySkan + 1;
	END_IF
	
	IF xInstalacjaHC1 THEN
		arModbusOdczytCykliczny[intPetlaPierwszySkan].bAdresUrzadzenia := bAdres;
		arModbusOdczytCykliczny[intPetlaPierwszySkan].bFunkcja := TO_BYTE(enumModbusKodyFunkcji.OdczytNRejestrowWejsciowych);
		arModbusOdczytCykliczny[intPetlaPierwszySkan].uiAdresRejestru := 400;
		arModbusOdczytCykliczny[intPetlaPierwszySkan].ltCzestotliwosc := TIME_TO_LTIME(tMinimalnyCzasRaportowania);
		arModbusOdczytCykliczny[intPetlaPierwszySkan].pZmiennaReferencyjna := ADR(wTrybPracyHC1);
		intPetlaPierwszySkan := intPetlaPierwszySkan + 1;
	END_IF
	
	IF xInstalacjaHC1 THEN
		arModbusOdczytCykliczny[intPetlaPierwszySkan].bAdresUrzadzenia := bAdres;
		arModbusOdczytCykliczny[intPetlaPierwszySkan].bFunkcja := TO_BYTE(enumModbusKodyFunkcji.OdczytNRejestrowWejsciowych);
		arModbusOdczytCykliczny[intPetlaPierwszySkan].uiAdresRejestru := 401;
		arModbusOdczytCykliczny[intPetlaPierwszySkan].ltCzestotliwosc := TIME_TO_LTIME(tMinimalnyCzasRaportowania);
		arModbusOdczytCykliczny[intPetlaPierwszySkan].pZmiennaReferencyjna := ADR(wTrybOperacjiHC1);
		intPetlaPierwszySkan := intPetlaPierwszySkan + 1;
	END_IF
	
	IF xInstalacjaHC1 THEN
		arModbusOdczytCykliczny[intPetlaPierwszySkan].bAdresUrzadzenia := bAdres;
		arModbusOdczytCykliczny[intPetlaPierwszySkan].bFunkcja := TO_BYTE(enumModbusKodyFunkcji.OdczytNRejestrowWejsciowych);
		arModbusOdczytCykliczny[intPetlaPierwszySkan].uiAdresRejestru := 419;
		arModbusOdczytCykliczny[intPetlaPierwszySkan].ltCzestotliwosc := TIME_TO_LTIME(tMinimalnyCzasRaportowania);
		arModbusOdczytCykliczny[intPetlaPierwszySkan].pZmiennaReferencyjna := ADR(wTemperaturaGrzaniaNastawionaHC1);
		intPetlaPierwszySkan := intPetlaPierwszySkan + 1;
	END_IF
		
	IF xInstalacjaHC1 THEN
		arModbusOdczytCykliczny[intPetlaPierwszySkan].bAdresUrzadzenia := bAdres;
		arModbusOdczytCykliczny[intPetlaPierwszySkan].bFunkcja := TO_BYTE(enumModbusKodyFunkcji.OdczytNRejestrowWejsciowych);
		arModbusOdczytCykliczny[intPetlaPierwszySkan].uiAdresRejestru := 420;
		arModbusOdczytCykliczny[intPetlaPierwszySkan].ltCzestotliwosc := TIME_TO_LTIME(tMinimalnyCzasRaportowania);
		arModbusOdczytCykliczny[intPetlaPierwszySkan].pZmiennaReferencyjna := ADR(wTemperaturaGrzaniaNastawionaKrzywaGrzewczaHC1);
		intPetlaPierwszySkan := intPetlaPierwszySkan + 1;
	END_IF

	IF xInstalacjaHC1 THEN
		arModbusOdczytCykliczny[intPetlaPierwszySkan].bAdresUrzadzenia := bAdres;
		arModbusOdczytCykliczny[intPetlaPierwszySkan].bFunkcja := TO_BYTE(enumModbusKodyFunkcji.OdczytNRejestrowWejsciowych);
		arModbusOdczytCykliczny[intPetlaPierwszySkan].uiAdresRejestru := 451;
		arModbusOdczytCykliczny[intPetlaPierwszySkan].ltCzestotliwosc := TIME_TO_LTIME(tMinimalnyCzasRaportowania);
		arModbusOdczytCykliczny[intPetlaPierwszySkan].pZmiennaReferencyjna := ADR(wTemperaturaPowrotuMiastoHC1);
		intPetlaPierwszySkan := intPetlaPierwszySkan + 1;
	END_IF
	
	IF xInstalacjaHC1 THEN
		arModbusOdczytCykliczny[intPetlaPierwszySkan].bAdresUrzadzenia := bAdres;
		arModbusOdczytCykliczny[intPetlaPierwszySkan].bFunkcja := TO_BYTE(enumModbusKodyFunkcji.OdczytNRejestrowWejsciowych);
		arModbusOdczytCykliczny[intPetlaPierwszySkan].uiAdresRejestru := 474;
		arModbusOdczytCykliczny[intPetlaPierwszySkan].ltCzestotliwosc := TIME_TO_LTIME(tMinimalnyCzasRaportowania);
		arModbusOdczytCykliczny[intPetlaPierwszySkan].pZmiennaReferencyjna := ADR(wSygnalZadaniaGrzaniaHC1);
		intPetlaPierwszySkan := intPetlaPierwszySkan + 1;
	END_IF
	
	IF xInstalacjaHC1 THEN
		arModbusOdczytCykliczny[intPetlaPierwszySkan].bAdresUrzadzenia := bAdres;
		arModbusOdczytCykliczny[intPetlaPierwszySkan].bFunkcja := TO_BYTE(enumModbusKodyFunkcji.OdczytNRejestrowWejsciowych);
		arModbusOdczytCykliczny[intPetlaPierwszySkan].uiAdresRejestru := 489;
		arModbusOdczytCykliczny[intPetlaPierwszySkan].ltCzestotliwosc := TIME_TO_LTIME(tMinimalnyCzasRaportowania);
		arModbusOdczytCykliczny[intPetlaPierwszySkan].pZmiennaReferencyjna := ADR(wStopienOtwarciaZaworuMiastoHC1);
		intPetlaPierwszySkan := intPetlaPierwszySkan + 1;
	END_IF
	
	IF xInstalacjaDHW THEN
		arModbusOdczytCykliczny[intPetlaPierwszySkan].bAdresUrzadzenia := bAdres;
		arModbusOdczytCykliczny[intPetlaPierwszySkan].bFunkcja := TO_BYTE(enumModbusKodyFunkcji.OdczytNRejestrowWejsciowych);
		arModbusOdczytCykliczny[intPetlaPierwszySkan].uiAdresRejestru := 800;
		arModbusOdczytCykliczny[intPetlaPierwszySkan].ltCzestotliwosc := TIME_TO_LTIME(tMinimalnyCzasRaportowania);
		arModbusOdczytCykliczny[intPetlaPierwszySkan].pZmiennaReferencyjna := ADR(wTrybPracyDHW);
		intPetlaPierwszySkan := intPetlaPierwszySkan + 1;
	END_IF
	
	IF xInstalacjaDHW THEN
		arModbusOdczytCykliczny[intPetlaPierwszySkan].bAdresUrzadzenia := bAdres;
		arModbusOdczytCykliczny[intPetlaPierwszySkan].bFunkcja := TO_BYTE(enumModbusKodyFunkcji.OdczytNRejestrowWejsciowych);
		arModbusOdczytCykliczny[intPetlaPierwszySkan].uiAdresRejestru := 801;
		arModbusOdczytCykliczny[intPetlaPierwszySkan].ltCzestotliwosc := TIME_TO_LTIME(tMinimalnyCzasRaportowania);
		arModbusOdczytCykliczny[intPetlaPierwszySkan].pZmiennaReferencyjna := ADR(wTrybOperacjiDHW);
		intPetlaPierwszySkan := intPetlaPierwszySkan + 1;
	END_IF
	
	IF xInstalacjaDHW THEN
		arModbusOdczytCykliczny[intPetlaPierwszySkan].bAdresUrzadzenia := bAdres;
		arModbusOdczytCykliczny[intPetlaPierwszySkan].bFunkcja := TO_BYTE(enumModbusKodyFunkcji.OdczytNRejestrowWejsciowych);
		arModbusOdczytCykliczny[intPetlaPierwszySkan].uiAdresRejestru := 819;
		arModbusOdczytCykliczny[intPetlaPierwszySkan].ltCzestotliwosc := TIME_TO_LTIME(tMinimalnyCzasRaportowania);
		arModbusOdczytCykliczny[intPetlaPierwszySkan].pZmiennaReferencyjna := ADR(wTemperaturaGrzaniaNastawionaDHW);
		intPetlaPierwszySkan := intPetlaPierwszySkan + 1;
	END_IF
	
	IF xInstalacjaDHW THEN
		arModbusOdczytCykliczny[intPetlaPierwszySkan].bAdresUrzadzenia := bAdres;
		arModbusOdczytCykliczny[intPetlaPierwszySkan].bFunkcja := TO_BYTE(enumModbusKodyFunkcji.OdczytNRejestrowWejsciowych);
		arModbusOdczytCykliczny[intPetlaPierwszySkan].uiAdresRejestru := 849;
		arModbusOdczytCykliczny[intPetlaPierwszySkan].ltCzestotliwosc := TIME_TO_LTIME(tMinimalnyCzasRaportowania);
		arModbusOdczytCykliczny[intPetlaPierwszySkan].pZmiennaReferencyjna := ADR(wTemperaturaZasilaniaBudynekDHW);
		intPetlaPierwszySkan := intPetlaPierwszySkan + 1;
	END_IF
	
	IF xInstalacjaDHW THEN
		arModbusOdczytCykliczny[intPetlaPierwszySkan].bAdresUrzadzenia := bAdres;
		arModbusOdczytCykliczny[intPetlaPierwszySkan].bFunkcja := TO_BYTE(enumModbusKodyFunkcji.OdczytNRejestrowWejsciowych);
		arModbusOdczytCykliczny[intPetlaPierwszySkan].uiAdresRejestru := 850;
		arModbusOdczytCykliczny[intPetlaPierwszySkan].ltCzestotliwosc := TIME_TO_LTIME(tMinimalnyCzasRaportowania);
		arModbusOdczytCykliczny[intPetlaPierwszySkan].pZmiennaReferencyjna := ADR(wTemperaturaPowrotuBudynekDHW);
		intPetlaPierwszySkan := intPetlaPierwszySkan + 1;
	END_IF
	
	IF xInstalacjaDHW THEN
		arModbusOdczytCykliczny[intPetlaPierwszySkan].bAdresUrzadzenia := bAdres;
		arModbusOdczytCykliczny[intPetlaPierwszySkan].bFunkcja := TO_BYTE(enumModbusKodyFunkcji.OdczytNRejestrowWejsciowych);
		arModbusOdczytCykliczny[intPetlaPierwszySkan].uiAdresRejestru := 854;
		arModbusOdczytCykliczny[intPetlaPierwszySkan].ltCzestotliwosc := TIME_TO_LTIME(tMinimalnyCzasRaportowania);
		arModbusOdczytCykliczny[intPetlaPierwszySkan].pZmiennaReferencyjna := ADR(wTemperaturaPowrotuMiastoDHW);
		intPetlaPierwszySkan := intPetlaPierwszySkan + 1;
	END_IF
	
	IF xInstalacjaDHW THEN
		arModbusOdczytCykliczny[intPetlaPierwszySkan].bAdresUrzadzenia := bAdres;
		arModbusOdczytCykliczny[intPetlaPierwszySkan].bFunkcja := TO_BYTE(enumModbusKodyFunkcji.OdczytNRejestrowWejsciowych);
		arModbusOdczytCykliczny[intPetlaPierwszySkan].uiAdresRejestru := 889;
		arModbusOdczytCykliczny[intPetlaPierwszySkan].ltCzestotliwosc := TIME_TO_LTIME(tMinimalnyCzasRaportowania);
		arModbusOdczytCykliczny[intPetlaPierwszySkan].pZmiennaReferencyjna := ADR(wStopienOtwarciaZaworuMiastoDHW);
		intPetlaPierwszySkan := intPetlaPierwszySkan + 1;
	END_IF
	
	//holding register	
	IF xInstalacjaHC1 THEN
		arModbusOdczytCykliczny[intPetlaPierwszySkan].bAdresUrzadzenia := bAdres;
		arModbusOdczytCykliczny[intPetlaPierwszySkan].bFunkcja := TO_BYTE(enumModbusKodyFunkcji.OdczytNRejestrow);
		arModbusOdczytCykliczny[intPetlaPierwszySkan].uiAdresRejestru := 424;
		arModbusOdczytCykliczny[intPetlaPierwszySkan].ltCzestotliwosc := TIME_TO_LTIME(tMinimalnyCzasRaportowania);
		arModbusOdczytCykliczny[intPetlaPierwszySkan].pZmiennaReferencyjna := ADR(wKrzywaGrzewczaTemperaturyZewnetrznejX2OdczytHC1);
		intPetlaPierwszySkan := intPetlaPierwszySkan + 1;
	END_IF
	
	IF xInstalacjaHC1 THEN
		arModbusOdczytCykliczny[intPetlaPierwszySkan].bAdresUrzadzenia := bAdres;
		arModbusOdczytCykliczny[intPetlaPierwszySkan].bFunkcja := TO_BYTE(enumModbusKodyFunkcji.OdczytNRejestrow);
		arModbusOdczytCykliczny[intPetlaPierwszySkan].uiAdresRejestru := 425;
		arModbusOdczytCykliczny[intPetlaPierwszySkan].ltCzestotliwosc := TIME_TO_LTIME(tMinimalnyCzasRaportowania);
		arModbusOdczytCykliczny[intPetlaPierwszySkan].pZmiennaReferencyjna := ADR(wKrzywaGrzewczaTemperaturyZewnetrznejX6OdczytHC1);
		intPetlaPierwszySkan := intPetlaPierwszySkan + 1;
	END_IF
	
	IF xInstalacjaHC1 THEN
		arModbusOdczytCykliczny[intPetlaPierwszySkan].bAdresUrzadzenia := bAdres;
		arModbusOdczytCykliczny[intPetlaPierwszySkan].bFunkcja := TO_BYTE(enumModbusKodyFunkcji.OdczytNRejestrow);
		arModbusOdczytCykliczny[intPetlaPierwszySkan].uiAdresRejestru := 426;
		arModbusOdczytCykliczny[intPetlaPierwszySkan].ltCzestotliwosc := TIME_TO_LTIME(tMinimalnyCzasRaportowania);
		arModbusOdczytCykliczny[intPetlaPierwszySkan].pZmiennaReferencyjna := ADR(wKrzywaGrzewczaTemperaturyZasilaniaY2OdczytHC1);
		intPetlaPierwszySkan := intPetlaPierwszySkan + 1;
	END_IF
	
	IF xInstalacjaHC1 THEN
		arModbusOdczytCykliczny[intPetlaPierwszySkan].bAdresUrzadzenia := bAdres;
		arModbusOdczytCykliczny[intPetlaPierwszySkan].bFunkcja := TO_BYTE(enumModbusKodyFunkcji.OdczytNRejestrow);
		arModbusOdczytCykliczny[intPetlaPierwszySkan].uiAdresRejestru := 427;
		arModbusOdczytCykliczny[intPetlaPierwszySkan].ltCzestotliwosc := TIME_TO_LTIME(tMinimalnyCzasRaportowania);
		arModbusOdczytCykliczny[intPetlaPierwszySkan].pZmiennaReferencyjna := ADR(wKrzywaGrzewczaTemperaturyZasilaniaY6OdczytHC1);
		intPetlaPierwszySkan := intPetlaPierwszySkan + 1;
	END_IF
	
	IF xInstalacjaHC1 THEN
		arModbusOdczytCykliczny[intPetlaPierwszySkan].bAdresUrzadzenia := bAdres;
		arModbusOdczytCykliczny[intPetlaPierwszySkan].bFunkcja := TO_BYTE(enumModbusKodyFunkcji.OdczytNRejestrow);
		arModbusOdczytCykliczny[intPetlaPierwszySkan].uiAdresRejestru := 435;
		arModbusOdczytCykliczny[intPetlaPierwszySkan].ltCzestotliwosc := TIME_TO_LTIME(tMinimalnyCzasRaportowania);
		arModbusOdczytCykliczny[intPetlaPierwszySkan].pZmiennaReferencyjna := ADR(wKrzywaGrzewczaTemperaturyZasilaniaY3OdczytHC1);
		intPetlaPierwszySkan := intPetlaPierwszySkan + 1;
	END_IF
	
	IF xInstalacjaHC1 THEN
		arModbusOdczytCykliczny[intPetlaPierwszySkan].bAdresUrzadzenia := bAdres;
		arModbusOdczytCykliczny[intPetlaPierwszySkan].bFunkcja := TO_BYTE(enumModbusKodyFunkcji.OdczytNRejestrow);
		arModbusOdczytCykliczny[intPetlaPierwszySkan].uiAdresRejestru := 436;
		arModbusOdczytCykliczny[intPetlaPierwszySkan].ltCzestotliwosc := TIME_TO_LTIME(tMinimalnyCzasRaportowania);
		arModbusOdczytCykliczny[intPetlaPierwszySkan].pZmiennaReferencyjna := ADR(wKrzywaGrzewczaTemperaturyZasilaniaY4OdczytHC1);
		intPetlaPierwszySkan := intPetlaPierwszySkan + 1;
	END_IF
	
	IF xInstalacjaHC1 THEN
		arModbusOdczytCykliczny[intPetlaPierwszySkan].bAdresUrzadzenia := bAdres;
		arModbusOdczytCykliczny[intPetlaPierwszySkan].bFunkcja := TO_BYTE(enumModbusKodyFunkcji.OdczytNRejestrow);
		arModbusOdczytCykliczny[intPetlaPierwszySkan].uiAdresRejestru := 437;
		arModbusOdczytCykliczny[intPetlaPierwszySkan].ltCzestotliwosc := TIME_TO_LTIME(tMinimalnyCzasRaportowania);
		arModbusOdczytCykliczny[intPetlaPierwszySkan].pZmiennaReferencyjna := ADR(wKrzywaGrzewczaTemperaturyZasilaniaY5OdczytHC1);
		intPetlaPierwszySkan := intPetlaPierwszySkan + 1;
	END_IF
	
	IF xInstalacjaHC1 THEN
		arModbusOdczytCykliczny[intPetlaPierwszySkan].bAdresUrzadzenia := bAdres;
		arModbusOdczytCykliczny[intPetlaPierwszySkan].bFunkcja := TO_BYTE(enumModbusKodyFunkcji.OdczytNRejestrow);
		arModbusOdczytCykliczny[intPetlaPierwszySkan].uiAdresRejestru := 449;
		arModbusOdczytCykliczny[intPetlaPierwszySkan].ltCzestotliwosc := TIME_TO_LTIME(tMinimalnyCzasRaportowania);
		arModbusOdczytCykliczny[intPetlaPierwszySkan].pZmiennaReferencyjna := ADR(wKrzywaGrzewczaTemperaturyZewnetrznejX3OdczytHC1);
		intPetlaPierwszySkan := intPetlaPierwszySkan + 1;
	END_IF
	
	IF xInstalacjaHC1 THEN
		arModbusOdczytCykliczny[intPetlaPierwszySkan].bAdresUrzadzenia := bAdres;
		arModbusOdczytCykliczny[intPetlaPierwszySkan].bFunkcja := TO_BYTE(enumModbusKodyFunkcji.OdczytNRejestrow);
		arModbusOdczytCykliczny[intPetlaPierwszySkan].uiAdresRejestru := 450;
		arModbusOdczytCykliczny[intPetlaPierwszySkan].ltCzestotliwosc := TIME_TO_LTIME(tMinimalnyCzasRaportowania);
		arModbusOdczytCykliczny[intPetlaPierwszySkan].pZmiennaReferencyjna := ADR(wKrzywaGrzewczaTemperaturyZewnetrznejX4OdczytHC1);
		intPetlaPierwszySkan := intPetlaPierwszySkan + 1;
	END_IF
	
	IF xInstalacjaHC1 THEN
		arModbusOdczytCykliczny[intPetlaPierwszySkan].bAdresUrzadzenia := bAdres;
		arModbusOdczytCykliczny[intPetlaPierwszySkan].bFunkcja := TO_BYTE(enumModbusKodyFunkcji.OdczytNRejestrow);
		arModbusOdczytCykliczny[intPetlaPierwszySkan].uiAdresRejestru := 451;
		arModbusOdczytCykliczny[intPetlaPierwszySkan].ltCzestotliwosc := TIME_TO_LTIME(tMinimalnyCzasRaportowania);
		arModbusOdczytCykliczny[intPetlaPierwszySkan].pZmiennaReferencyjna := ADR(wKrzywaGrzewczaTemperaturyZewnetrznejX5OdczytHC1);
		intPetlaPierwszySkan := intPetlaPierwszySkan + 1;
	END_IF
END_IF

//obsluga komunikatu przychodzacego z IZE

IF sKomunikat <> sKomunikatPamiec AND xPoInicjalizacji THEN
	sKomunikatPamiec := sKomunikat;
	IF fnIDOdbiorcyMatch(sKomunikat , sIdInstancji) THEN
		sDane := '';
		//rozkaz typu C
		IF fnKomunikatTyp(sKomunikat) = 'C' AND NOT xAutonomizacja THEN
			IF fnKomunikatDaneSzukajWartosci(sKomunikat,'BLOK=') = '0' THEN
				IF intBlokadaWykonywaniaRozkazow = 1 THEN
					intBlokadaWykonywaniaRozkazow := 0;
					xRaport := TRUE;
					ELSE	
					IF sDane <> '' THEN
					sDane := CONCAT(sDane , ';');
					END_IF
					sDane := CONCAT(sDane , 'BLOK=0');
				END_IF
			END_IF
			IF fnKomunikatDaneSzukajWartosci(sKomunikat,'BLOK=') = '1' THEN
				IF intBlokadaWykonywaniaRozkazow = 0 THEN
					intBlokadaWykonywaniaRozkazow := 1;
					xRaport := TRUE;
					ELSE
					IF sDane <> '' THEN
					sDane := CONCAT(sDane , ';');
					END_IF					
					sDane := CONCAT(sDane , 'BLOK=1');
				END_IF
			END_IF
			//sprawdzanie atrybutow dedykowanych dla urzadzenia - przygotowywanie do zapisu do Modbusa
			IF intBlokadaWykonywaniaRozkazow = 0 THEN
				// Tryb pracy HC1
				fnKomunikatDaneZnajdzPorownajZapisz(sKomunikat := sKomunikat,
					sAtrybut := 'TRYBNASHC1=',
					rAtrybutWartosc := rTrybPracyHC1Zapis,
					sDane := sDane,
					xAtrybutZapisz => xTrybPracyHC1Zapisz);	
				// Temperatura punktu X2 krzywej grzewczej HC1
				fnKomunikatDaneZnajdzPorownajZapisz(sKomunikat := sKomunikat,
					sAtrybut := 'TEMPKGHC1X2=',
					rAtrybutWartosc := rKrzywaGrzewczaTemperaturyZewnetrznejX2HC1Zapis,
					sDane := sDane,
					xAtrybutZapisz => xKrzywaGrzewczaTemperaturyZewnetrznejX2HC1Zapisz);
				// Temperatura punktu X3 krzywej grzewczej HC1
				fnKomunikatDaneZnajdzPorownajZapisz(sKomunikat := sKomunikat,
					sAtrybut := 'TEMPKGHC1X3=',
					rAtrybutWartosc := rKrzywaGrzewczaTemperaturyZewnetrznejX3HC1Zapis,
					sDane := sDane,
					xAtrybutZapisz => xKrzywaGrzewczaTemperaturyZewnetrznejX3HC1Zapisz);
				// Temperatura punktu X4 krzywej grzewczej HC1
				fnKomunikatDaneZnajdzPorownajZapisz(sKomunikat := sKomunikat,
					sAtrybut := 'TEMPKGHC1X4=',
					rAtrybutWartosc := rKrzywaGrzewczaTemperaturyZewnetrznejX4HC1Zapis,
					sDane := sDane,
					xAtrybutZapisz => xKrzywaGrzewczaTemperaturyZewnetrznejX4HC1Zapisz);
				// Temperatura punktu X5 krzywej grzewczej HC1
				fnKomunikatDaneZnajdzPorownajZapisz(sKomunikat := sKomunikat,
					sAtrybut := 'TEMPKGHC1X5=',
					rAtrybutWartosc := rKrzywaGrzewczaTemperaturyZewnetrznejX5HC1Zapis,
					sDane := sDane,
					xAtrybutZapisz => xKrzywaGrzewczaTemperaturyZewnetrznejX5HC1Zapisz);
				// Temperatura punktu X6 krzywej grzewczej HC1
				fnKomunikatDaneZnajdzPorownajZapisz(sKomunikat := sKomunikat,
					sAtrybut := 'TEMPKGHC1X6=',
					rAtrybutWartosc := rKrzywaGrzewczaTemperaturyZewnetrznejX6HC1Zapis,
					sDane := sDane,
					xAtrybutZapisz => xKrzywaGrzewczaTemperaturyZewnetrznejX6HC1Zapisz);					
				// Temperatura punktu Y2 krzywej grzewczej HC1
				fnKomunikatDaneZnajdzPorownajZapisz(sKomunikat := sKomunikat,
					sAtrybut := 'TEMPKGHC1Y2=',
					rAtrybutWartosc := rKrzywaGrzewczaTemperaturyZasilaniaY2HC1Zapis,
					sDane := sDane,
					xAtrybutZapisz => xKrzywaGrzewczaTemperaturyZasilaniaY2HC1Zapisz);				
				// Temperatura punktu Y3 krzywej grzewczej HC1
				fnKomunikatDaneZnajdzPorownajZapisz(sKomunikat := sKomunikat,
					sAtrybut := 'TEMPKGHC1Y3=',
					rAtrybutWartosc := rKrzywaGrzewczaTemperaturyZasilaniaY3HC1Zapis,
					sDane := sDane,
					xAtrybutZapisz => xKrzywaGrzewczaTemperaturyZasilaniaY3HC1Zapisz);				
				// Temperatura punktu Y4 krzywej grzewczej HC1
				fnKomunikatDaneZnajdzPorownajZapisz(sKomunikat := sKomunikat,
					sAtrybut := 'TEMPKGHC1Y4=',
					rAtrybutWartosc := rKrzywaGrzewczaTemperaturyZasilaniaY4HC1Zapis,
					sDane := sDane,
					xAtrybutZapisz => xKrzywaGrzewczaTemperaturyZasilaniaY4HC1Zapisz);				
				// Temperatura punktu Y5 krzywej grzewczej HC1
				fnKomunikatDaneZnajdzPorownajZapisz(sKomunikat := sKomunikat,
					sAtrybut := 'TEMPKGHC1Y5=',
					rAtrybutWartosc := rKrzywaGrzewczaTemperaturyZasilaniaY5HC1Zapis,
					sDane := sDane,
					xAtrybutZapisz => xKrzywaGrzewczaTemperaturyZasilaniaY5HC1Zapisz);				
				// Temperatura punktu Y6 krzywej grzewczej HC1
				fnKomunikatDaneZnajdzPorownajZapisz(sKomunikat := sKomunikat,
					sAtrybut := 'TEMPKGHC1Y6=',
					rAtrybutWartosc := rKrzywaGrzewczaTemperaturyZasilaniaY6HC1Zapis,
					sDane := sDane,
					xAtrybutZapisz => xKrzywaGrzewczaTemperaturyZasilaniaY6HC1Zapisz);	
				// Tryb pracy DHW
				fnKomunikatDaneZnajdzPorownajZapisz(sKomunikat := sKomunikat,
					sAtrybut := 'TRYBNASDHW=',
					rAtrybutWartosc := rTrybPracyDHWZapis,
					sDane := sDane,
					xAtrybutZapisz => xTrybPracyDHWZapisz);	
			END_IF
		END_IF
				
		//raportowanie typu A na potwierdzanie stanow zadanych przez C
		IF sDane <> '' THEN
			fnZapiszKomunikat(	sCalyKomunikat := '' ,
								sTypKomunikatu := 'A' ,
								sMnemonik := sMnemonik ,
								sMACAdres := sMACAdres ,
								sIDNadawcy := sIdInstancji ,
								sIDOdbiorcy := sIdAplikacji ,
								sDaneZapasowe := sDaneZapasowe ,
								sDane := sDane ,
								arTablicaKomunikatow := arTablicaKomunikatow ,
								intTablicaKomunikatowZnacznikZapisu := intTablicaKomunikatowZnacznikZapisu ,
								intTablicaKomunikatowRozmiar := intTablicaKomunikatowRozmiar ,
								sWyslanyKomunikat := sWyslanyKomunikatDummy);
		END_IF
		
		sDane := '';
		//zapytanie typu Q
		IF fnKomunikatTyp(sKomunikat) = 'Q' AND arModbusStatusKomunikacji[bAdres] = enumModbusStatus.KomunikacjaPrawidlowa THEN
			IF fnKomunikatDaneSzukajWartosci(sKomunikat , 'BLOK=') = '?' OR fnKomunikatDaneSzukajWartosci(sKomunikat , 'ALL=') = '?' THEN
				fnKomunikatDaneDodaj_xOverFlow(sDane := sDane , sAtrybut := 'BLOK=' , sWartosc := INT_TO_STRING(intBlokadaWykonywaniaRozkazow) , xOverFlow := xOverFlow);	
				IF xOverFlow = TRUE THEN
					fnZapiszKomunikat(	sCalyKomunikat := '' ,
								sTypKomunikatu := 'A' ,
								sMnemonik := sMnemonik ,
								sMACAdres := sMACAdres ,
								sIDNadawcy := sIdInstancji ,
								sIDOdbiorcy := sIdAplikacji ,
								sDaneZapasowe := sDaneZapasowe ,
								sDane := sDane ,
								arTablicaKomunikatow := arTablicaKomunikatow ,
								intTablicaKomunikatowZnacznikZapisu := intTablicaKomunikatowZnacznikZapisu ,
								intTablicaKomunikatowRozmiar := intTablicaKomunikatowRozmiar ,
								sWyslanyKomunikat := sWyslanyKomunikatDummy);
					sDane := '';
				END_IF	
			END_IF
			IF xInstalacjaHC1 THEN
				IF fnKomunikatDaneSzukajWartosci(sKomunikat , 'TEMPZEW=') = '?' OR fnKomunikatDaneSzukajWartosci(sKomunikat , 'ALL=') = '?' THEN
					fnKomunikatDaneDodaj_xOverFlow(sDane := sDane , sAtrybut := 'TEMPZEW=' , sWartosc := REAL_TO_STRING(rTemperaturaZewnetrzna) , xOverFlow := xOverFlow);	
					IF xOverFlow = TRUE THEN
						fnZapiszKomunikat(	sCalyKomunikat := '' ,
									sTypKomunikatu := 'A' ,
									sMnemonik := sMnemonik ,
									sMACAdres := sMACAdres ,
									sIDNadawcy := sIdInstancji ,
									sIDOdbiorcy := sIdAplikacji ,
									sDaneZapasowe := sDaneZapasowe ,
									sDane := sDane ,
									arTablicaKomunikatow := arTablicaKomunikatow ,
									intTablicaKomunikatowZnacznikZapisu := intTablicaKomunikatowZnacznikZapisu ,
									intTablicaKomunikatowRozmiar := intTablicaKomunikatowRozmiar ,
									sWyslanyKomunikat := sWyslanyKomunikatDummy);
						sDane := '';
					END_IF	
				END_IF
				IF fnKomunikatDaneSzukajWartosci(sKomunikat , 'TEMPNASHC1=') = '?' OR fnKomunikatDaneSzukajWartosci(sKomunikat , 'ALL=') = '?' THEN
					fnKomunikatDaneDodaj_xOverFlow(sDane := sDane , sAtrybut := 'TEMPNASHC1=' , sWartosc := REAL_TO_STRING(rTemperaturaGrzaniaNastawionaHC1) , xOverFlow := xOverFlow);	
					IF xOverFlow = TRUE THEN
						fnZapiszKomunikat(	sCalyKomunikat := '' ,
									sTypKomunikatu := 'A' ,
									sMnemonik := sMnemonik ,
									sMACAdres := sMACAdres ,
									sIDNadawcy := sIdInstancji ,
									sIDOdbiorcy := sIdAplikacji ,
									sDaneZapasowe := sDaneZapasowe ,
									sDane := sDane ,
									arTablicaKomunikatow := arTablicaKomunikatow ,
									intTablicaKomunikatowZnacznikZapisu := intTablicaKomunikatowZnacznikZapisu ,
									intTablicaKomunikatowRozmiar := intTablicaKomunikatowRozmiar ,
									sWyslanyKomunikat := sWyslanyKomunikatDummy);
						sDane := '';
					END_IF	
				END_IF
				IF fnKomunikatDaneSzukajWartosci(sKomunikat , 'TEMPNASKGHC1=') = '?' OR fnKomunikatDaneSzukajWartosci(sKomunikat , 'ALL=') = '?' THEN
					fnKomunikatDaneDodaj_xOverFlow(sDane := sDane , sAtrybut := 'TEMPNASKGHC1=' , sWartosc := REAL_TO_STRING(rTemperaturaGrzaniaNastawionaKrzywaGrzewczaHC1) , xOverFlow := xOverFlow);	
					IF xOverFlow = TRUE THEN
						fnZapiszKomunikat(	sCalyKomunikat := '' ,
									sTypKomunikatu := 'A' ,
									sMnemonik := sMnemonik ,
									sMACAdres := sMACAdres ,
									sIDNadawcy := sIdInstancji ,
									sIDOdbiorcy := sIdAplikacji ,
									sDaneZapasowe := sDaneZapasowe ,
									sDane := sDane ,
									arTablicaKomunikatow := arTablicaKomunikatow ,
									intTablicaKomunikatowZnacznikZapisu := intTablicaKomunikatowZnacznikZapisu ,
									intTablicaKomunikatowRozmiar := intTablicaKomunikatowRozmiar ,
									sWyslanyKomunikat := sWyslanyKomunikatDummy);
						sDane := '';
					END_IF	
				END_IF
				IF fnKomunikatDaneSzukajWartosci(sKomunikat , 'TRYBNASHC1=') = '?' OR fnKomunikatDaneSzukajWartosci(sKomunikat , 'ALL=') = '?' THEN
					fnKomunikatDaneDodaj_xOverFlow(sDane := sDane , sAtrybut := 'TRYBNASHC1=' , sWartosc := INT_TO_STRING(intTrybPracyHC1) , xOverFlow := xOverFlow);	
					IF xOverFlow = TRUE THEN
						fnZapiszKomunikat(	sCalyKomunikat := '' ,
									sTypKomunikatu := 'A' ,
									sMnemonik := sMnemonik ,
									sMACAdres := sMACAdres ,
									sIDNadawcy := sIdInstancji ,
									sIDOdbiorcy := sIdAplikacji ,
									sDaneZapasowe := sDaneZapasowe ,
									sDane := sDane ,
									arTablicaKomunikatow := arTablicaKomunikatow ,
									intTablicaKomunikatowZnacznikZapisu := intTablicaKomunikatowZnacznikZapisu ,
									intTablicaKomunikatowRozmiar := intTablicaKomunikatowRozmiar ,
									sWyslanyKomunikat := sWyslanyKomunikatDummy);
						sDane := '';
					END_IF	
				END_IF
				IF fnKomunikatDaneSzukajWartosci(sKomunikat , 'TRYBOPHC1=') = '?' OR fnKomunikatDaneSzukajWartosci(sKomunikat , 'ALL=') = '?' THEN
					fnKomunikatDaneDodaj_xOverFlow(sDane := sDane , sAtrybut := 'TRYBOPHC1=' , sWartosc := INT_TO_STRING(intTrybOperacjiHC1) , xOverFlow := xOverFlow);	
					IF xOverFlow = TRUE THEN
						fnZapiszKomunikat(	sCalyKomunikat := '' ,
									sTypKomunikatu := 'A' ,
									sMnemonik := sMnemonik ,
									sMACAdres := sMACAdres ,
									sIDNadawcy := sIdInstancji ,
									sIDOdbiorcy := sIdAplikacji ,
									sDaneZapasowe := sDaneZapasowe ,
									sDane := sDane ,
									arTablicaKomunikatow := arTablicaKomunikatow ,
									intTablicaKomunikatowZnacznikZapisu := intTablicaKomunikatowZnacznikZapisu ,
									intTablicaKomunikatowRozmiar := intTablicaKomunikatowRozmiar ,
									sWyslanyKomunikat := sWyslanyKomunikatDummy);
						sDane := '';
					END_IF	
				END_IF
				IF fnKomunikatDaneSzukajWartosci(sKomunikat , 'TEMPZASOHC1=') = '?' OR fnKomunikatDaneSzukajWartosci(sKomunikat , 'ALL=') = '?' THEN
					fnKomunikatDaneDodaj_xOverFlow(sDane := sDane , sAtrybut := 'TEMPZASOHC1=' , sWartosc := REAL_TO_STRING(rTemperaturaZasilaniaObwoduHC1) , xOverFlow := xOverFlow);	
					IF xOverFlow = TRUE THEN
						fnZapiszKomunikat(	sCalyKomunikat := '' ,
									sTypKomunikatu := 'A' ,
									sMnemonik := sMnemonik ,
									sMACAdres := sMACAdres ,
									sIDNadawcy := sIdInstancji ,
									sIDOdbiorcy := sIdAplikacji ,
									sDaneZapasowe := sDaneZapasowe ,
									sDane := sDane ,
									arTablicaKomunikatow := arTablicaKomunikatow ,
									intTablicaKomunikatowZnacznikZapisu := intTablicaKomunikatowZnacznikZapisu ,
									intTablicaKomunikatowRozmiar := intTablicaKomunikatowRozmiar ,
									sWyslanyKomunikat := sWyslanyKomunikatDummy);
						sDane := '';
					END_IF	
				END_IF
				IF fnKomunikatDaneSzukajWartosci(sKomunikat , 'TEMPPOWOHC1=') = '?' OR fnKomunikatDaneSzukajWartosci(sKomunikat , 'ALL=') = '?' THEN
					fnKomunikatDaneDodaj_xOverFlow(sDane := sDane , sAtrybut := 'TEMPPOWOHC1=' , sWartosc := REAL_TO_STRING(rTemperaturaPowrotuObwoduHC1) , xOverFlow := xOverFlow);	
					IF xOverFlow = TRUE THEN
						fnZapiszKomunikat(	sCalyKomunikat := '' ,
									sTypKomunikatu := 'A' ,
									sMnemonik := sMnemonik ,
									sMACAdres := sMACAdres ,
									sIDNadawcy := sIdInstancji ,
									sIDOdbiorcy := sIdAplikacji ,
									sDaneZapasowe := sDaneZapasowe ,
									sDane := sDane ,
									arTablicaKomunikatow := arTablicaKomunikatow ,
									intTablicaKomunikatowZnacznikZapisu := intTablicaKomunikatowZnacznikZapisu ,
									intTablicaKomunikatowRozmiar := intTablicaKomunikatowRozmiar ,
									sWyslanyKomunikat := sWyslanyKomunikatDummy);
						sDane := '';
					END_IF	
				END_IF
				IF fnKomunikatDaneSzukajWartosci(sKomunikat , 'TEMPPOWMHC1=') = '?' OR fnKomunikatDaneSzukajWartosci(sKomunikat , 'ALL=') = '?' THEN
					fnKomunikatDaneDodaj_xOverFlow(sDane := sDane , sAtrybut := 'TEMPPOWMHC1=' , sWartosc := REAL_TO_STRING(rTemperaturaPowrotuMiastoHC1) , xOverFlow := xOverFlow);	
					IF xOverFlow = TRUE THEN
						fnZapiszKomunikat(	sCalyKomunikat := '' ,
									sTypKomunikatu := 'A' ,
									sMnemonik := sMnemonik ,
									sMACAdres := sMACAdres ,
									sIDNadawcy := sIdInstancji ,
									sIDOdbiorcy := sIdAplikacji ,
									sDaneZapasowe := sDaneZapasowe ,
									sDane := sDane ,
									arTablicaKomunikatow := arTablicaKomunikatow ,
									intTablicaKomunikatowZnacznikZapisu := intTablicaKomunikatowZnacznikZapisu ,
									intTablicaKomunikatowRozmiar := intTablicaKomunikatowRozmiar ,
									sWyslanyKomunikat := sWyslanyKomunikatDummy);
						sDane := '';
					END_IF	
				END_IF
				IF fnKomunikatDaneSzukajWartosci(sKomunikat , 'TEMPZASB=') = '?' OR fnKomunikatDaneSzukajWartosci(sKomunikat , 'ALL=') = '?' THEN
					fnKomunikatDaneDodaj_xOverFlow(sDane := sDane , sAtrybut := 'TEMPZASB=' , sWartosc := REAL_TO_STRING(rTemperaturaZasilaniaBudynku) , xOverFlow := xOverFlow);	
					IF xOverFlow = TRUE THEN
						fnZapiszKomunikat(	sCalyKomunikat := '' ,
									sTypKomunikatu := 'A' ,
									sMnemonik := sMnemonik ,
									sMACAdres := sMACAdres ,
									sIDNadawcy := sIdInstancji ,
									sIDOdbiorcy := sIdAplikacji ,
									sDaneZapasowe := sDaneZapasowe ,
									sDane := sDane ,
									arTablicaKomunikatow := arTablicaKomunikatow ,
									intTablicaKomunikatowZnacznikZapisu := intTablicaKomunikatowZnacznikZapisu ,
									intTablicaKomunikatowRozmiar := intTablicaKomunikatowRozmiar ,
									sWyslanyKomunikat := sWyslanyKomunikatDummy);
						sDane := '';
					END_IF	
				END_IF
				IF fnKomunikatDaneSzukajWartosci(sKomunikat , 'TEMPPOWB=') = '?' OR fnKomunikatDaneSzukajWartosci(sKomunikat , 'ALL=') = '?' THEN
					fnKomunikatDaneDodaj_xOverFlow(sDane := sDane , sAtrybut := 'TEMPPOWB=' , sWartosc := REAL_TO_STRING(rTemperaturaPowrotuBudynku) , xOverFlow := xOverFlow);	
					IF xOverFlow = TRUE THEN
						fnZapiszKomunikat(	sCalyKomunikat := '' ,
									sTypKomunikatu := 'A' ,
									sMnemonik := sMnemonik ,
									sMACAdres := sMACAdres ,
									sIDNadawcy := sIdInstancji ,
									sIDOdbiorcy := sIdAplikacji ,
									sDaneZapasowe := sDaneZapasowe ,
									sDane := sDane ,
									arTablicaKomunikatow := arTablicaKomunikatow ,
									intTablicaKomunikatowZnacznikZapisu := intTablicaKomunikatowZnacznikZapisu ,
									intTablicaKomunikatowRozmiar := intTablicaKomunikatowRozmiar ,
									sWyslanyKomunikat := sWyslanyKomunikatDummy);
						sDane := '';
					END_IF	
				END_IF
				IF fnKomunikatDaneSzukajWartosci(sKomunikat , 'STERGRZHC1=') = '?' OR fnKomunikatDaneSzukajWartosci(sKomunikat , 'ALL=') = '?' THEN
					fnKomunikatDaneDodaj_xOverFlow(sDane := sDane , sAtrybut := 'STERGRZHC1=' , sWartosc := REAL_TO_STRING(rSygnalZadaniaGrzaniaHC1) , xOverFlow := xOverFlow);	
					IF xOverFlow = TRUE THEN
						fnZapiszKomunikat(	sCalyKomunikat := '' ,
									sTypKomunikatu := 'A' ,
									sMnemonik := sMnemonik ,
									sMACAdres := sMACAdres ,
									sIDNadawcy := sIdInstancji ,
									sIDOdbiorcy := sIdAplikacji ,
									sDaneZapasowe := sDaneZapasowe ,
									sDane := sDane ,
									arTablicaKomunikatow := arTablicaKomunikatow ,
									intTablicaKomunikatowZnacznikZapisu := intTablicaKomunikatowZnacznikZapisu ,
									intTablicaKomunikatowRozmiar := intTablicaKomunikatowRozmiar ,
									sWyslanyKomunikat := sWyslanyKomunikatDummy);
						sDane := '';
					END_IF	
				END_IF
				IF fnKomunikatDaneSzukajWartosci(sKomunikat , 'STERZAWMHC1=') = '?' OR fnKomunikatDaneSzukajWartosci(sKomunikat , 'ALL=') = '?' THEN
					fnKomunikatDaneDodaj_xOverFlow(sDane := sDane , sAtrybut := 'STERZAWMHC1=' , sWartosc := REAL_TO_STRING(rStopienOtwarciaZaworuMiastoHC1) , xOverFlow := xOverFlow);	
					IF xOverFlow = TRUE THEN
						fnZapiszKomunikat(	sCalyKomunikat := '' ,
									sTypKomunikatu := 'A' ,
									sMnemonik := sMnemonik ,
									sMACAdres := sMACAdres ,
									sIDNadawcy := sIdInstancji ,
									sIDOdbiorcy := sIdAplikacji ,
									sDaneZapasowe := sDaneZapasowe ,
									sDane := sDane ,
									arTablicaKomunikatow := arTablicaKomunikatow ,
									intTablicaKomunikatowZnacznikZapisu := intTablicaKomunikatowZnacznikZapisu ,
									intTablicaKomunikatowRozmiar := intTablicaKomunikatowRozmiar ,
									sWyslanyKomunikat := sWyslanyKomunikatDummy);
						sDane := '';
					END_IF	
				END_IF
				IF fnKomunikatDaneSzukajWartosci(sKomunikat , 'TEMPKGHC1X2=') = '?' OR fnKomunikatDaneSzukajWartosci(sKomunikat , 'ALL=') = '?' THEN
					fnKomunikatDaneDodaj_xOverFlow(sDane := sDane , sAtrybut := 'TEMPKGHC1X2=' , sWartosc := REAL_TO_STRING(rKrzywaGrzewczaTemperaturyZewnetrznejX2HC1) , xOverFlow := xOverFlow);	
					IF xOverFlow = TRUE THEN
						fnZapiszKomunikat(	sCalyKomunikat := '' ,
									sTypKomunikatu := 'A' ,
									sMnemonik := sMnemonik ,
									sMACAdres := sMACAdres ,
									sIDNadawcy := sIdInstancji ,
									sIDOdbiorcy := sIdAplikacji ,
									sDaneZapasowe := sDaneZapasowe ,
									sDane := sDane ,
									arTablicaKomunikatow := arTablicaKomunikatow ,
									intTablicaKomunikatowZnacznikZapisu := intTablicaKomunikatowZnacznikZapisu ,
									intTablicaKomunikatowRozmiar := intTablicaKomunikatowRozmiar ,
									sWyslanyKomunikat := sWyslanyKomunikatDummy);
						sDane := '';
					END_IF
				END_IF
				IF fnKomunikatDaneSzukajWartosci(sKomunikat , 'TEMPKGHC1X3=') = '?' OR fnKomunikatDaneSzukajWartosci(sKomunikat , 'ALL=') = '?' THEN
					fnKomunikatDaneDodaj_xOverFlow(sDane := sDane , sAtrybut := 'TEMPKGHC1X3=' , sWartosc := REAL_TO_STRING(rKrzywaGrzewczaTemperaturyZewnetrznejX3HC1) , xOverFlow := xOverFlow);	
					IF xOverFlow = TRUE THEN
						fnZapiszKomunikat(	sCalyKomunikat := '' ,
									sTypKomunikatu := 'A' ,
									sMnemonik := sMnemonik ,
									sMACAdres := sMACAdres ,
									sIDNadawcy := sIdInstancji ,
									sIDOdbiorcy := sIdAplikacji ,
									sDaneZapasowe := sDaneZapasowe ,
									sDane := sDane ,
									arTablicaKomunikatow := arTablicaKomunikatow ,
									intTablicaKomunikatowZnacznikZapisu := intTablicaKomunikatowZnacznikZapisu ,
									intTablicaKomunikatowRozmiar := intTablicaKomunikatowRozmiar ,
									sWyslanyKomunikat := sWyslanyKomunikatDummy);
						sDane := '';
					END_IF
				END_IF
				IF fnKomunikatDaneSzukajWartosci(sKomunikat , 'TEMPKGHC1X4=') = '?' OR fnKomunikatDaneSzukajWartosci(sKomunikat , 'ALL=') = '?' THEN
					fnKomunikatDaneDodaj_xOverFlow(sDane := sDane , sAtrybut := 'TEMPKGHC1X4=' , sWartosc := REAL_TO_STRING(rKrzywaGrzewczaTemperaturyZewnetrznejX4HC1) , xOverFlow := xOverFlow);	
					IF xOverFlow = TRUE THEN
						fnZapiszKomunikat(	sCalyKomunikat := '' ,
									sTypKomunikatu := 'A' ,
									sMnemonik := sMnemonik ,
									sMACAdres := sMACAdres ,
									sIDNadawcy := sIdInstancji ,
									sIDOdbiorcy := sIdAplikacji ,
									sDaneZapasowe := sDaneZapasowe ,
									sDane := sDane ,
									arTablicaKomunikatow := arTablicaKomunikatow ,
									intTablicaKomunikatowZnacznikZapisu := intTablicaKomunikatowZnacznikZapisu ,
									intTablicaKomunikatowRozmiar := intTablicaKomunikatowRozmiar ,
									sWyslanyKomunikat := sWyslanyKomunikatDummy);
						sDane := '';
					END_IF
				END_IF
				IF fnKomunikatDaneSzukajWartosci(sKomunikat , 'TEMPKGHC1X5=') = '?' OR fnKomunikatDaneSzukajWartosci(sKomunikat , 'ALL=') = '?' THEN
					fnKomunikatDaneDodaj_xOverFlow(sDane := sDane , sAtrybut := 'TEMPKGHC1X5=' , sWartosc := REAL_TO_STRING(rKrzywaGrzewczaTemperaturyZewnetrznejX5HC1) , xOverFlow := xOverFlow);	
					IF xOverFlow = TRUE THEN
						fnZapiszKomunikat(	sCalyKomunikat := '' ,
									sTypKomunikatu := 'A' ,
									sMnemonik := sMnemonik ,
									sMACAdres := sMACAdres ,
									sIDNadawcy := sIdInstancji ,
									sIDOdbiorcy := sIdAplikacji ,
									sDaneZapasowe := sDaneZapasowe ,
									sDane := sDane ,
									arTablicaKomunikatow := arTablicaKomunikatow ,
									intTablicaKomunikatowZnacznikZapisu := intTablicaKomunikatowZnacznikZapisu ,
									intTablicaKomunikatowRozmiar := intTablicaKomunikatowRozmiar ,
									sWyslanyKomunikat := sWyslanyKomunikatDummy);
						sDane := '';
					END_IF
				END_IF
				IF fnKomunikatDaneSzukajWartosci(sKomunikat , 'TEMPKGHC1X6=') = '?' OR fnKomunikatDaneSzukajWartosci(sKomunikat , 'ALL=') = '?' THEN
					fnKomunikatDaneDodaj_xOverFlow(sDane := sDane , sAtrybut := 'TEMPKGHC1X6=' , sWartosc := REAL_TO_STRING(rKrzywaGrzewczaTemperaturyZewnetrznejX6HC1) , xOverFlow := xOverFlow);	
					IF xOverFlow = TRUE THEN
						fnZapiszKomunikat(	sCalyKomunikat := '' ,
									sTypKomunikatu := 'A' ,
									sMnemonik := sMnemonik ,
									sMACAdres := sMACAdres ,
									sIDNadawcy := sIdInstancji ,
									sIDOdbiorcy := sIdAplikacji ,
									sDaneZapasowe := sDaneZapasowe ,
									sDane := sDane ,
									arTablicaKomunikatow := arTablicaKomunikatow ,
									intTablicaKomunikatowZnacznikZapisu := intTablicaKomunikatowZnacznikZapisu ,
									intTablicaKomunikatowRozmiar := intTablicaKomunikatowRozmiar ,
									sWyslanyKomunikat := sWyslanyKomunikatDummy);
						sDane := '';
					END_IF
				END_IF
				IF fnKomunikatDaneSzukajWartosci(sKomunikat , 'TEMPKGHC1Y2=') = '?' OR fnKomunikatDaneSzukajWartosci(sKomunikat , 'ALL=') = '?' THEN
					fnKomunikatDaneDodaj_xOverFlow(sDane := sDane , sAtrybut := 'TEMPKGHC1Y2=' , sWartosc := REAL_TO_STRING(rKrzywaGrzewczaTemperaturyZasilaniaY2HC1) , xOverFlow := xOverFlow);	
					IF xOverFlow = TRUE THEN
						fnZapiszKomunikat(	sCalyKomunikat := '' ,
									sTypKomunikatu := 'A' ,
									sMnemonik := sMnemonik ,
									sMACAdres := sMACAdres ,
									sIDNadawcy := sIdInstancji ,
									sIDOdbiorcy := sIdAplikacji ,
									sDaneZapasowe := sDaneZapasowe ,
									sDane := sDane ,
									arTablicaKomunikatow := arTablicaKomunikatow ,
									intTablicaKomunikatowZnacznikZapisu := intTablicaKomunikatowZnacznikZapisu ,
									intTablicaKomunikatowRozmiar := intTablicaKomunikatowRozmiar ,
									sWyslanyKomunikat := sWyslanyKomunikatDummy);
						sDane := '';
					END_IF
				END_IF
				IF fnKomunikatDaneSzukajWartosci(sKomunikat , 'TEMPKGHC1Y3=') = '?' OR fnKomunikatDaneSzukajWartosci(sKomunikat , 'ALL=') = '?' THEN
					fnKomunikatDaneDodaj_xOverFlow(sDane := sDane , sAtrybut := 'TEMPKGHC1Y3=' , sWartosc := REAL_TO_STRING(rKrzywaGrzewczaTemperaturyZasilaniaY3HC1) , xOverFlow := xOverFlow);	
					IF xOverFlow = TRUE THEN
						fnZapiszKomunikat(	sCalyKomunikat := '' ,
									sTypKomunikatu := 'A' ,
									sMnemonik := sMnemonik ,
									sMACAdres := sMACAdres ,
									sIDNadawcy := sIdInstancji ,
									sIDOdbiorcy := sIdAplikacji ,
									sDaneZapasowe := sDaneZapasowe ,
									sDane := sDane ,
									arTablicaKomunikatow := arTablicaKomunikatow ,
									intTablicaKomunikatowZnacznikZapisu := intTablicaKomunikatowZnacznikZapisu ,
									intTablicaKomunikatowRozmiar := intTablicaKomunikatowRozmiar ,
									sWyslanyKomunikat := sWyslanyKomunikatDummy);
						sDane := '';
					END_IF
				END_IF
				IF fnKomunikatDaneSzukajWartosci(sKomunikat , 'TEMPKGHC1Y4=') = '?' OR fnKomunikatDaneSzukajWartosci(sKomunikat , 'ALL=') = '?' THEN
					fnKomunikatDaneDodaj_xOverFlow(sDane := sDane , sAtrybut := 'TEMPKGHC1Y4=' , sWartosc := REAL_TO_STRING(rKrzywaGrzewczaTemperaturyZasilaniaY4HC1) , xOverFlow := xOverFlow);	
					IF xOverFlow = TRUE THEN
						fnZapiszKomunikat(	sCalyKomunikat := '' ,
									sTypKomunikatu := 'A' ,
									sMnemonik := sMnemonik ,
									sMACAdres := sMACAdres ,
									sIDNadawcy := sIdInstancji ,
									sIDOdbiorcy := sIdAplikacji ,
									sDaneZapasowe := sDaneZapasowe ,
									sDane := sDane ,
									arTablicaKomunikatow := arTablicaKomunikatow ,
									intTablicaKomunikatowZnacznikZapisu := intTablicaKomunikatowZnacznikZapisu ,
									intTablicaKomunikatowRozmiar := intTablicaKomunikatowRozmiar ,
									sWyslanyKomunikat := sWyslanyKomunikatDummy);
						sDane := '';
					END_IF
				END_IF
				IF fnKomunikatDaneSzukajWartosci(sKomunikat , 'TEMPKGHC1Y5=') = '?' OR fnKomunikatDaneSzukajWartosci(sKomunikat , 'ALL=') = '?' THEN
					fnKomunikatDaneDodaj_xOverFlow(sDane := sDane , sAtrybut := 'TEMPKGHC1Y5=' , sWartosc := REAL_TO_STRING(rKrzywaGrzewczaTemperaturyZasilaniaY5HC1) , xOverFlow := xOverFlow);	
					IF xOverFlow = TRUE THEN
						fnZapiszKomunikat(	sCalyKomunikat := '' ,
									sTypKomunikatu := 'A' ,
									sMnemonik := sMnemonik ,
									sMACAdres := sMACAdres ,
									sIDNadawcy := sIdInstancji ,
									sIDOdbiorcy := sIdAplikacji ,
									sDaneZapasowe := sDaneZapasowe ,
									sDane := sDane ,
									arTablicaKomunikatow := arTablicaKomunikatow ,
									intTablicaKomunikatowZnacznikZapisu := intTablicaKomunikatowZnacznikZapisu ,
									intTablicaKomunikatowRozmiar := intTablicaKomunikatowRozmiar ,
									sWyslanyKomunikat := sWyslanyKomunikatDummy);
						sDane := '';
					END_IF
				END_IF
				IF fnKomunikatDaneSzukajWartosci(sKomunikat , 'TEMPKGHC1Y6=') = '?' OR fnKomunikatDaneSzukajWartosci(sKomunikat , 'ALL=') = '?' THEN
					fnKomunikatDaneDodaj_xOverFlow(sDane := sDane , sAtrybut := 'TEMPKGHC1Y6=' , sWartosc := REAL_TO_STRING(rKrzywaGrzewczaTemperaturyZasilaniaY6HC1) , xOverFlow := xOverFlow);	
					IF xOverFlow = TRUE THEN
						fnZapiszKomunikat(	sCalyKomunikat := '' ,
									sTypKomunikatu := 'A' ,
									sMnemonik := sMnemonik ,
									sMACAdres := sMACAdres ,
									sIDNadawcy := sIdInstancji ,
									sIDOdbiorcy := sIdAplikacji ,
									sDaneZapasowe := sDaneZapasowe ,
									sDane := sDane ,
									arTablicaKomunikatow := arTablicaKomunikatow ,
									intTablicaKomunikatowZnacznikZapisu := intTablicaKomunikatowZnacznikZapisu ,
									intTablicaKomunikatowRozmiar := intTablicaKomunikatowRozmiar ,
									sWyslanyKomunikat := sWyslanyKomunikatDummy);
						sDane := '';
					END_IF
				END_IF
				IF fnKomunikatDaneSzukajWartosci(sKomunikat , 'SEZONGRZ=') = '?' OR fnKomunikatDaneSzukajWartosci(sKomunikat , 'ALL=') = '?' THEN
					fnKomunikatDaneDodaj_xOverFlow(sDane := sDane , sAtrybut := 'SEZONGRZ=' , sWartosc := BOOL_TO_STRING(xSezonGrzewczy) , xOverFlow := xOverFlow);	
					IF xOverFlow = TRUE THEN
						fnZapiszKomunikat(	sCalyKomunikat := '' ,
									sTypKomunikatu := 'A' ,
									sMnemonik := sMnemonik ,
									sMACAdres := sMACAdres ,
									sIDNadawcy := sIdInstancji ,
									sIDOdbiorcy := sIdAplikacji ,
									sDaneZapasowe := sDaneZapasowe ,
									sDane := sDane ,
									arTablicaKomunikatow := arTablicaKomunikatow ,
									intTablicaKomunikatowZnacznikZapisu := intTablicaKomunikatowZnacznikZapisu ,
									intTablicaKomunikatowRozmiar := intTablicaKomunikatowRozmiar ,
									sWyslanyKomunikat := sWyslanyKomunikatDummy);
						sDane := '';
					END_IF
				END_IF
				IF fnKomunikatDaneSzukajWartosci(sKomunikat , 'TEMPSR1DZ=') = '?' OR fnKomunikatDaneSzukajWartosci(sKomunikat , 'ALL=') = '?' THEN
					fnKomunikatDaneDodaj_xOverFlow(sDane := sDane , sAtrybut := 'TEMPSR1DZ=' , sWartosc := REAL_TO_STRING(rTemperaturaSrednia1Dzien + 273.15) , xOverFlow := xOverFlow);	
					IF xOverFlow = TRUE THEN
						fnZapiszKomunikat(	sCalyKomunikat := '' ,
									sTypKomunikatu := 'A' ,
									sMnemonik := sMnemonik ,
									sMACAdres := sMACAdres ,
									sIDNadawcy := sIdInstancji ,
									sIDOdbiorcy := sIdAplikacji ,
									sDaneZapasowe := sDaneZapasowe ,
									sDane := sDane ,
									arTablicaKomunikatow := arTablicaKomunikatow ,
									intTablicaKomunikatowZnacznikZapisu := intTablicaKomunikatowZnacznikZapisu ,
									intTablicaKomunikatowRozmiar := intTablicaKomunikatowRozmiar ,
									sWyslanyKomunikat := sWyslanyKomunikatDummy);
						sDane := '';
					END_IF
				END_IF				
			END_IF
			IF xInstalacjaDHW THEN
				IF fnKomunikatDaneSzukajWartosci(sKomunikat , 'TEMPNASDHW=') = '?' OR fnKomunikatDaneSzukajWartosci(sKomunikat , 'ALL=') = '?' THEN
					fnKomunikatDaneDodaj_xOverFlow(sDane := sDane , sAtrybut := 'TEMPNASDHW=' , sWartosc := REAL_TO_STRING(rTemperaturaGrzaniaNastawionaDHW) , xOverFlow := xOverFlow);	
					IF xOverFlow = TRUE THEN
						fnZapiszKomunikat(	sCalyKomunikat := '' ,
									sTypKomunikatu := 'A' ,
									sMnemonik := sMnemonik ,
									sMACAdres := sMACAdres ,
									sIDNadawcy := sIdInstancji ,
									sIDOdbiorcy := sIdAplikacji ,
									sDaneZapasowe := sDaneZapasowe ,
									sDane := sDane ,
									arTablicaKomunikatow := arTablicaKomunikatow ,
									intTablicaKomunikatowZnacznikZapisu := intTablicaKomunikatowZnacznikZapisu ,
									intTablicaKomunikatowRozmiar := intTablicaKomunikatowRozmiar ,
									sWyslanyKomunikat := sWyslanyKomunikatDummy);
						sDane := '';
					END_IF
				END_IF
				IF fnKomunikatDaneSzukajWartosci(sKomunikat , 'TRYBNASDHW=') = '?' OR fnKomunikatDaneSzukajWartosci(sKomunikat , 'ALL=') = '?' THEN
					fnKomunikatDaneDodaj_xOverFlow(sDane := sDane , sAtrybut := 'TRYBNASDHW=' , sWartosc := INT_TO_STRING(intTrybPracyDHW) , xOverFlow := xOverFlow);	
					IF xOverFlow = TRUE THEN
						fnZapiszKomunikat(	sCalyKomunikat := '' ,
									sTypKomunikatu := 'A' ,
									sMnemonik := sMnemonik ,
									sMACAdres := sMACAdres ,
									sIDNadawcy := sIdInstancji ,
									sIDOdbiorcy := sIdAplikacji ,
									sDaneZapasowe := sDaneZapasowe ,
									sDane := sDane ,
									arTablicaKomunikatow := arTablicaKomunikatow ,
									intTablicaKomunikatowZnacznikZapisu := intTablicaKomunikatowZnacznikZapisu ,
									intTablicaKomunikatowRozmiar := intTablicaKomunikatowRozmiar ,
									sWyslanyKomunikat := sWyslanyKomunikatDummy);
						sDane := '';
					END_IF	
				END_IF
				IF fnKomunikatDaneSzukajWartosci(sKomunikat , 'TRYBOPDHW=') = '?' OR fnKomunikatDaneSzukajWartosci(sKomunikat , 'ALL=') = '?' THEN
					fnKomunikatDaneDodaj_xOverFlow(sDane := sDane , sAtrybut := 'TRYBOPDHW=' , sWartosc := INT_TO_STRING(intTrybOperacjiDHW) , xOverFlow := xOverFlow);	
					IF xOverFlow = TRUE THEN
						fnZapiszKomunikat(	sCalyKomunikat := '' ,
									sTypKomunikatu := 'A' ,
									sMnemonik := sMnemonik ,
									sMACAdres := sMACAdres ,
									sIDNadawcy := sIdInstancji ,
									sIDOdbiorcy := sIdAplikacji ,
									sDaneZapasowe := sDaneZapasowe ,
									sDane := sDane ,
									arTablicaKomunikatow := arTablicaKomunikatow ,
									intTablicaKomunikatowZnacznikZapisu := intTablicaKomunikatowZnacznikZapisu ,
									intTablicaKomunikatowRozmiar := intTablicaKomunikatowRozmiar ,
									sWyslanyKomunikat := sWyslanyKomunikatDummy);
						sDane := '';
					END_IF	
				END_IF
				IF fnKomunikatDaneSzukajWartosci(sKomunikat , 'TEMPPOWMDHW=') = '?' OR fnKomunikatDaneSzukajWartosci(sKomunikat , 'ALL=') = '?' THEN
					fnKomunikatDaneDodaj_xOverFlow(sDane := sDane , sAtrybut := 'TEMPPOWMDHW=' , sWartosc := REAL_TO_STRING(rTemperaturaPowrotuMiastoDHW) , xOverFlow := xOverFlow);	
					IF xOverFlow = TRUE THEN
						fnZapiszKomunikat(	sCalyKomunikat := '' ,
									sTypKomunikatu := 'A' ,
									sMnemonik := sMnemonik ,
									sMACAdres := sMACAdres ,
									sIDNadawcy := sIdInstancji ,
									sIDOdbiorcy := sIdAplikacji ,
									sDaneZapasowe := sDaneZapasowe ,
									sDane := sDane ,
									arTablicaKomunikatow := arTablicaKomunikatow ,
									intTablicaKomunikatowZnacznikZapisu := intTablicaKomunikatowZnacznikZapisu ,
									intTablicaKomunikatowRozmiar := intTablicaKomunikatowRozmiar ,
									sWyslanyKomunikat := sWyslanyKomunikatDummy);
						sDane := '';
					END_IF
				END_IF
				IF fnKomunikatDaneSzukajWartosci(sKomunikat , 'TEMPZASBDHW=') = '?' OR fnKomunikatDaneSzukajWartosci(sKomunikat , 'ALL=') = '?' THEN
					fnKomunikatDaneDodaj_xOverFlow(sDane := sDane , sAtrybut := 'TEMPZASBDHW=' , sWartosc := REAL_TO_STRING(rTemperaturaZasilaniaBudynekDHW) , xOverFlow := xOverFlow);	
					IF xOverFlow = TRUE THEN
						fnZapiszKomunikat(	sCalyKomunikat := '' ,
									sTypKomunikatu := 'A' ,
									sMnemonik := sMnemonik ,
									sMACAdres := sMACAdres ,
									sIDNadawcy := sIdInstancji ,
									sIDOdbiorcy := sIdAplikacji ,
									sDaneZapasowe := sDaneZapasowe ,
									sDane := sDane ,
									arTablicaKomunikatow := arTablicaKomunikatow ,
									intTablicaKomunikatowZnacznikZapisu := intTablicaKomunikatowZnacznikZapisu ,
									intTablicaKomunikatowRozmiar := intTablicaKomunikatowRozmiar ,
									sWyslanyKomunikat := sWyslanyKomunikatDummy);
						sDane := '';
					END_IF
				END_IF
				IF fnKomunikatDaneSzukajWartosci(sKomunikat , 'TEMPPOWBDHW=') = '?' OR fnKomunikatDaneSzukajWartosci(sKomunikat , 'ALL=') = '?' THEN
					fnKomunikatDaneDodaj_xOverFlow(sDane := sDane , sAtrybut := 'TEMPPOWBDHW=' , sWartosc := REAL_TO_STRING(rTemperaturaPowrotuBudynekDHW) , xOverFlow := xOverFlow);	
					IF xOverFlow = TRUE THEN
						fnZapiszKomunikat(	sCalyKomunikat := '' ,
									sTypKomunikatu := 'A' ,
									sMnemonik := sMnemonik ,
									sMACAdres := sMACAdres ,
									sIDNadawcy := sIdInstancji ,
									sIDOdbiorcy := sIdAplikacji ,
									sDaneZapasowe := sDaneZapasowe ,
									sDane := sDane ,
									arTablicaKomunikatow := arTablicaKomunikatow ,
									intTablicaKomunikatowZnacznikZapisu := intTablicaKomunikatowZnacznikZapisu ,
									intTablicaKomunikatowRozmiar := intTablicaKomunikatowRozmiar ,
									sWyslanyKomunikat := sWyslanyKomunikatDummy);
						sDane := '';
					END_IF
				END_IF
				IF fnKomunikatDaneSzukajWartosci(sKomunikat , 'STERZAWMDHW=') = '?' OR fnKomunikatDaneSzukajWartosci(sKomunikat , 'ALL=') = '?' THEN
					fnKomunikatDaneDodaj_xOverFlow(sDane := sDane , sAtrybut := 'STERZAWMDHW=' , sWartosc := REAL_TO_STRING(rStopienOtwarciaZaworuMiastoDHW) , xOverFlow := xOverFlow);	
					IF xOverFlow = TRUE THEN
						fnZapiszKomunikat(	sCalyKomunikat := '' ,
									sTypKomunikatu := 'A' ,
									sMnemonik := sMnemonik ,
									sMACAdres := sMACAdres ,
									sIDNadawcy := sIdInstancji ,
									sIDOdbiorcy := sIdAplikacji ,
									sDaneZapasowe := sDaneZapasowe ,
									sDane := sDane ,
									arTablicaKomunikatow := arTablicaKomunikatow ,
									intTablicaKomunikatowZnacznikZapisu := intTablicaKomunikatowZnacznikZapisu ,
									intTablicaKomunikatowRozmiar := intTablicaKomunikatowRozmiar ,
									sWyslanyKomunikat := sWyslanyKomunikatDummy);
						sDane := '';
					END_IF
				END_IF
			END_IF
			//pytanie o stany alarmów
			IF fnKomunikatDaneSzukajWartosci(sKomunikat , 'ALARM=') = '?' OR fnKomunikatDaneSzukajWartosci(sKomunikat , 'ALL=') = '?' THEN
				FOR intPetla := 1 TO 11 BY 1 DO
					//raportowanie typu E (stanów alarmów) na zapytanie typu Q
					IF arErrorStan[intPetla] <> enumAlarmWartosc.StanNieznany THEN
						fnZapiszKomunikat(	sCalyKomunikat := '' ,
											sTypKomunikatu := 'E' ,
											sMnemonik := sMnemonik ,
											sMACAdres := sMACAdres ,
											sIDNadawcy := sIdInstancji ,
											sIDOdbiorcy := sIdAplikacji ,
											sDaneZapasowe := sDaneZapasowe ,
											sDane := fnKomunikatDaneErrorRetry(xAktywny := arErrorStan[intPetla] = enumAlarmWartosc.StanAlarmowy , intKlasa := arErrorKlasa[intPetla] , intNumer := intPetla),
											arTablicaKomunikatow := arTablicaKomunikatow ,
											intTablicaKomunikatowZnacznikZapisu := intTablicaKomunikatowZnacznikZapisu ,
											intTablicaKomunikatowRozmiar := intTablicaKomunikatowRozmiar ,
											sWyslanyKomunikat := sWyslanyKomunikatDummy);
					END_IF
				END_FOR
			END_IF
		END_IF
		//raportowanie typu A na zapytanie Q
		IF sDane <> '' THEN
			fnZapiszKomunikat(	sCalyKomunikat := '' ,
								sTypKomunikatu := 'A' ,
								sMnemonik := sMnemonik ,
								sMACAdres := sMACAdres ,
								sIDNadawcy := sIdInstancji ,
								sIDOdbiorcy := sIdAplikacji ,
								sDaneZapasowe := sDaneZapasowe ,
								sDane := sDane ,
								arTablicaKomunikatow := arTablicaKomunikatow ,
								intTablicaKomunikatowZnacznikZapisu := intTablicaKomunikatowZnacznikZapisu ,
								intTablicaKomunikatowRozmiar := intTablicaKomunikatowRozmiar ,
								sWyslanyKomunikat := sWyslanyKomunikatDummy);
		END_IF
	END_IF
END_IF

// Przywrócenie wartości domyślnych nastaw krzywej grzewczej i trybów pracy w przypadku restartu sterownika lub przejścia w stan autonomizacji (brak komunikacji z IZE)
rtrigPrzywrocDomyslne(CLK := xAutonomizacja);
IF rtrigPrzywrocDomyslne.Q THEN	
	IF intTrybPracyHC1 <> intTrybPracyHC1Autonomizacja THEN
		rTrybPracyHC1Zapis := INT_TO_REAL(intTrybPracyHC1Autonomizacja);
		xTrybPracyHC1Zapisz := TRUE;
	END_IF
	IF rKrzywaGrzewczaTemperaturyZewnetrznejX2HC1 <> rKrzywaGrzewczaTemperaturyZewnetrznejX2HC1Autonomizacja THEN
		rKrzywaGrzewczaTemperaturyZewnetrznejX2HC1Zapis := rKrzywaGrzewczaTemperaturyZewnetrznejX2HC1Autonomizacja;
		xKrzywaGrzewczaTemperaturyZewnetrznejX2HC1Zapisz := TRUE;
	END_IF
	IF rKrzywaGrzewczaTemperaturyZewnetrznejX3HC1 <> rKrzywaGrzewczaTemperaturyZewnetrznejX3HC1Autonomizacja THEN
		rKrzywaGrzewczaTemperaturyZewnetrznejX3HC1Zapis := rKrzywaGrzewczaTemperaturyZewnetrznejX3HC1Autonomizacja;
		xKrzywaGrzewczaTemperaturyZewnetrznejX3HC1Zapisz := TRUE;
	END_IF
	IF rKrzywaGrzewczaTemperaturyZewnetrznejX4HC1 <> rKrzywaGrzewczaTemperaturyZewnetrznejX4HC1Autonomizacja THEN
		rKrzywaGrzewczaTemperaturyZewnetrznejX4HC1Zapis := rKrzywaGrzewczaTemperaturyZewnetrznejX4HC1Autonomizacja;
		xKrzywaGrzewczaTemperaturyZewnetrznejX4HC1Zapisz := TRUE;
	END_IF
	IF rKrzywaGrzewczaTemperaturyZewnetrznejX5HC1 <> rKrzywaGrzewczaTemperaturyZewnetrznejX5HC1Autonomizacja THEN
		rKrzywaGrzewczaTemperaturyZewnetrznejX5HC1Zapis := rKrzywaGrzewczaTemperaturyZewnetrznejX5HC1Autonomizacja;
		xKrzywaGrzewczaTemperaturyZewnetrznejX5HC1Zapisz := TRUE;
	END_IF
	IF rKrzywaGrzewczaTemperaturyZewnetrznejX6HC1 <> rKrzywaGrzewczaTemperaturyZewnetrznejX6HC1Autonomizacja THEN
		rKrzywaGrzewczaTemperaturyZewnetrznejX6HC1Zapis := rKrzywaGrzewczaTemperaturyZewnetrznejX6HC1Autonomizacja;
		xKrzywaGrzewczaTemperaturyZewnetrznejX6HC1Zapisz := TRUE;
	END_IF
	IF rKrzywaGrzewczaTemperaturyZasilaniaY2HC1 <> rKrzywaGrzewczaTemperaturyZasilaniaY2HC1Autonomizacja THEN
		rKrzywaGrzewczaTemperaturyZasilaniaY2HC1Zapis := rKrzywaGrzewczaTemperaturyZasilaniaY2HC1Autonomizacja;
		xKrzywaGrzewczaTemperaturyZasilaniaY2HC1Zapisz := TRUE;
	END_IF
	IF rKrzywaGrzewczaTemperaturyZasilaniaY3HC1 <> rKrzywaGrzewczaTemperaturyZasilaniaY3HC1Autonomizacja THEN
		rKrzywaGrzewczaTemperaturyZasilaniaY3HC1Zapis := rKrzywaGrzewczaTemperaturyZasilaniaY3HC1Autonomizacja;
		xKrzywaGrzewczaTemperaturyZasilaniaY3HC1Zapisz := TRUE;
	END_IF
	IF rKrzywaGrzewczaTemperaturyZasilaniaY4HC1 <> rKrzywaGrzewczaTemperaturyZasilaniaY4HC1Autonomizacja THEN
		rKrzywaGrzewczaTemperaturyZasilaniaY4HC1Zapis := rKrzywaGrzewczaTemperaturyZasilaniaY4HC1Autonomizacja;
		xKrzywaGrzewczaTemperaturyZasilaniaY4HC1Zapisz := TRUE;
	END_IF
	IF rKrzywaGrzewczaTemperaturyZasilaniaY5HC1 <> rKrzywaGrzewczaTemperaturyZasilaniaY5HC1Autonomizacja THEN
		rKrzywaGrzewczaTemperaturyZasilaniaY5HC1Zapis := rKrzywaGrzewczaTemperaturyZasilaniaY5HC1Autonomizacja;
		xKrzywaGrzewczaTemperaturyZasilaniaY5HC1Zapisz := TRUE;
	END_IF
	IF rKrzywaGrzewczaTemperaturyZasilaniaY6HC1 <> rKrzywaGrzewczaTemperaturyZasilaniaY6HC1Autonomizacja THEN
		rKrzywaGrzewczaTemperaturyZasilaniaY6HC1Zapis := rKrzywaGrzewczaTemperaturyZasilaniaY6HC1Autonomizacja;
		xKrzywaGrzewczaTemperaturyZasilaniaY6HC1Zapisz := TRUE;
	END_IF
	IF intTrybPracyDHW <> intTrybPracyDHWAutonomizacja THEN
		rTrybPracyDHWZapis := INT_TO_REAL(intTrybPracyDHWAutonomizacja);
		xTrybPracyDHWZapisz := TRUE;
	END_IF
END_IF	

// Trigger zapisu po Modbusie
rtrigZapisModbus (CLK := 	xTrybPracyHC1Zapisz OR xKrzywaGrzewczaTemperaturyZewnetrznejX2HC1Zapisz OR xKrzywaGrzewczaTemperaturyZewnetrznejX3HC1Zapisz OR xKrzywaGrzewczaTemperaturyZewnetrznejX4HC1Zapisz OR
							xKrzywaGrzewczaTemperaturyZewnetrznejX5HC1Zapisz OR xKrzywaGrzewczaTemperaturyZewnetrznejX6HC1Zapisz OR xKrzywaGrzewczaTemperaturyZasilaniaY2HC1Zapisz OR 
							xKrzywaGrzewczaTemperaturyZasilaniaY3HC1Zapisz OR xKrzywaGrzewczaTemperaturyZasilaniaY4HC1Zapisz OR xKrzywaGrzewczaTemperaturyZasilaniaY5HC1Zapisz OR
							xKrzywaGrzewczaTemperaturyZasilaniaY6HC1Zapisz OR xTrybPracyDHWZapisz);

// Taktowanie zapisywania po Modbusie
fbTaktowanieZapisywaniaModbus(IN := NOT fbTaktowanieZapisywaniaModbus.Q, PT := T#180S);
				
